   instHMISettings.instAsnBtnPrms.settings.stations.nextGroup.animate := 4;
   instHMISettings.instAsnBtnPrms.settings.stations.prevGroup.animate := 4;
   instHMISettings.instAsnBtnPrms.settings.stations.selectBtns[0].animate := 4;
   instHMISettings.instAsnBtnPrms.settings.stations.selectBtns[0].label := WSTRING#'1BX 3.0 1';
   instHMISettings.instAsnBtnPrms.settings.stations.selectBtns[1].animate := 4;
   instHMISettings.instAsnBtnPrms.settings.stations.selectBtns[1].label := WSTRING#'1BX 3.0 2';
   instHMISettings.instAsnBtnPrms.settings.stations.selectBtns[2].animate := 4;
   instHMISettings.instAsnBtnPrms.settings.stations.selectBtns[2].label := WSTRING#'1BX 3.0 3';
   instHMISettings.instAsnBtnPrms.settings.stations.selectBtns[3].animate := 4;
   instHMISettings.instAsnBtnPrms.settings.stations.selectBtns[3].label := WSTRING#'VOLVO 16 1';
   instHMISettings.instAsnBtnPrms.settings.stations.selectBtns[4].animate := 4;
   instHMISettings.instAsnBtnPrms.settings.stations.selectBtns[4].label := WSTRING#'VOLVO 16 2';
   instHMISettings.instAsnBtnPrms.settings.stations.selectBtns[5].animate := 4;
   instHMISettings.instAsnBtnPrms.settings.stations.selectBtns[5].label := WSTRING#'VOLVO 16 3';
   instHMISettings.instAsnBtnPrms.settings.stations.selectBtns[6].animate := 4;
   instHMISettings.instAsnBtnPrms.settings.stations.selectBtns[6].label := WSTRING#'VOLVO 16 4';
   instHMISettings.instAsnBtnPrms.settings.stations.selectBtns[7].animate := 4;
   instHMISettings.instAsnBtnPrms.settings.stations.selectBtns[7].label := WSTRING#'VOLVO 16 5';
   instHMISettings.instAsnBtnPrms.settings.stations.selectBtns[8].animate := 4;
   instHMISettings.instAsnBtnPrms.settings.stations.selectBtns[8].label := WSTRING#'VOLVO 16 6';
   instHMISettings.instAsnBtnPrms.settings.stations.selectBtns[9].animate := 4;
   instHMISettings.instAsnBtnPrms.settings.stations.selectBtns[9].label := WSTRING#'VOLVO 16 7';
   instHMISettings.instAsnBtnPrms.settings.stations.selectBtns[10].animate := 4;
   instHMISettings.instAsnBtnPrms.settings.stations.selectBtns[10].label := WSTRING#'VOLVO 16 8';
   instHMISettings.instAsnBtnPrms.settings.stations.selectBtns[11].animate := 4;
   instHMISettings.instAsnBtnPrms.settings.stations.selectBtns[11].label := WSTRING#'VOLVO 16 9';
   instHMISettings.instAsnBtnPrms.settings.stations.selCount := 1;
   instHMISettings.instAsnBtnPrms.settings.stations.selNumber := 19;
   instHMISettings.instAsnBtnPrms.settings.partNumber.assign.animate := 254;
   instHMISettings.instAsnBtnPrms.settings.partNumber.assign.label := WSTRING#'';
   instHMISettings.instAsnBtnPrms.settings.partNumber.ioField.animate := 254;
   instHMISettings.instAsnBtnPrms.settings.partNumber.ioField.inputFinished := TRUE;
   instHMISettings.instAsnBtnPrms.settings.partNumber.ioField.value := WSTRING#'';
   instHMISettings.instAsnBtnPrms.settings.viewingStation.btns[0].alloted.animate := 4;
   instHMISettings.instAsnBtnPrms.settings.viewingStation.btns[0].alloted.value := WSTRING#'30:00';
   instHMISettings.instAsnBtnPrms.settings.viewingStation.btns[0].critical.animate := 4;
   instHMISettings.instAsnBtnPrms.settings.viewingStation.btns[0].critical.value := WSTRING#'05:00';
   instHMISettings.instAsnBtnPrms.settings.viewingStation.btns[0].label.animate := 4;
   instHMISettings.instAsnBtnPrms.settings.viewingStation.btns[0].label.value := WSTRING#'1';
   instHMISettings.instAsnBtnPrms.settings.viewingStation.btns[0].partNumber.animate := 4;
   instHMISettings.instAsnBtnPrms.settings.viewingStation.btns[0].partNumber.value := WSTRING#'16.08.211.511.020F';
   instHMISettings.instAsnBtnPrms.settings.viewingStation.btns[1].alloted.animate := 4;
   instHMISettings.instAsnBtnPrms.settings.viewingStation.btns[1].alloted.value := WSTRING#'30:00';
   instHMISettings.instAsnBtnPrms.settings.viewingStation.btns[1].critical.animate := 4;
   instHMISettings.instAsnBtnPrms.settings.viewingStation.btns[1].critical.value := WSTRING#'05:00';
   instHMISettings.instAsnBtnPrms.settings.viewingStation.btns[1].label.animate := 4;
   instHMISettings.instAsnBtnPrms.settings.viewingStation.btns[1].label.value := WSTRING#'2';
   instHMISettings.instAsnBtnPrms.settings.viewingStation.btns[1].partNumber.animate := 4;
   instHMISettings.instAsnBtnPrms.settings.viewingStation.btns[1].partNumber.value := WSTRING#'16.08.208.151.010F';
   instHMISettings.instAsnBtnPrms.settings.viewingStation.btns[2].alloted.animate := 4;
   instHMISettings.instAsnBtnPrms.settings.viewingStation.btns[2].alloted.value := WSTRING#'30:00';
   instHMISettings.instAsnBtnPrms.settings.viewingStation.btns[2].critical.animate := 4;
   instHMISettings.instAsnBtnPrms.settings.viewingStation.btns[2].critical.value := WSTRING#'05:00';
   instHMISettings.instAsnBtnPrms.settings.viewingStation.btns[2].label.animate := 4;
   instHMISettings.instAsnBtnPrms.settings.viewingStation.btns[2].label.value := WSTRING#'3';
   instHMISettings.instAsnBtnPrms.settings.viewingStation.btns[2].partNumber.animate := 4;
   instHMISettings.instAsnBtnPrms.settings.viewingStation.btns[2].partNumber.value := WSTRING#'16.08.216.151.010B';
   instHMISettings.instAsnBtnPrms.settings.viewingStation.btns[3].alloted.animate := 4;
   instHMISettings.instAsnBtnPrms.settings.viewingStation.btns[3].alloted.value := WSTRING#'30:00';
   instHMISettings.instAsnBtnPrms.settings.viewingStation.btns[3].critical.animate := 4;
   instHMISettings.instAsnBtnPrms.settings.viewingStation.btns[3].critical.value := WSTRING#'05:00';
   instHMISettings.instAsnBtnPrms.settings.viewingStation.btns[3].label.animate := 4;
   instHMISettings.instAsnBtnPrms.settings.viewingStation.btns[3].label.value := WSTRING#'4';
   instHMISettings.instAsnBtnPrms.settings.viewingStation.btns[3].partNumber.animate := 4;
   instHMISettings.instAsnBtnPrms.settings.viewingStation.btns[3].partNumber.value := WSTRING#'16.08.216.831.020A';
   instHMISettings.instAsnBtnPrms.settings.viewingStation.btns[4].alloted.animate := 4;
   instHMISettings.instAsnBtnPrms.settings.viewingStation.btns[4].alloted.value := WSTRING#'02:00';
   instHMISettings.instAsnBtnPrms.settings.viewingStation.btns[4].critical.animate := 4;
   instHMISettings.instAsnBtnPrms.settings.viewingStation.btns[4].critical.value := WSTRING#'01:10';
   instHMISettings.instAsnBtnPrms.settings.viewingStation.btns[4].label.animate := 4;
   instHMISettings.instAsnBtnPrms.settings.viewingStation.btns[4].label.value := WSTRING#'5';
   instHMISettings.instAsnBtnPrms.settings.viewingStation.btns[4].partNumber.animate := 4;
   instHMISettings.instAsnBtnPrms.settings.viewingStation.btns[4].partNumber.value := WSTRING#'16.08.217.411.080A';
   instHMISettings.instAsnBtnPrms.settings.viewingStation.btns[5].alloted.animate := 4;
   instHMISettings.instAsnBtnPrms.settings.viewingStation.btns[5].alloted.value := WSTRING#'30:00';
   instHMISettings.instAsnBtnPrms.settings.viewingStation.btns[5].critical.animate := 4;
   instHMISettings.instAsnBtnPrms.settings.viewingStation.btns[5].critical.value := WSTRING#'05:00';
   instHMISettings.instAsnBtnPrms.settings.viewingStation.btns[5].label.animate := 4;
   instHMISettings.instAsnBtnPrms.settings.viewingStation.btns[5].label.value := WSTRING#'6';
   instHMISettings.instAsnBtnPrms.settings.viewingStation.btns[5].partNumber.animate := 4;
   instHMISettings.instAsnBtnPrms.settings.viewingStation.btns[5].partNumber.value := WSTRING#'16.08.216.521.000F';
   instHMISettings.instAsnBtnPrms.settings.viewingStation.btns[6].alloted.animate := 4;
   instHMISettings.instAsnBtnPrms.settings.viewingStation.btns[6].alloted.value := WSTRING#'00:00';
   instHMISettings.instAsnBtnPrms.settings.viewingStation.btns[6].critical.animate := 4;
   instHMISettings.instAsnBtnPrms.settings.viewingStation.btns[6].critical.value := WSTRING#'00:00';
   instHMISettings.instAsnBtnPrms.settings.viewingStation.btns[6].label.animate := 4;
   instHMISettings.instAsnBtnPrms.settings.viewingStation.btns[6].label.value := WSTRING#'7';
   instHMISettings.instAsnBtnPrms.settings.viewingStation.btns[6].partNumber.animate := 4;
   instHMISettings.instAsnBtnPrms.settings.viewingStation.btns[6].partNumber.value := WSTRING#'';
   instHMISettings.instAsnBtnPrms.settings.viewingStation.btns[7].alloted.animate := 4;
   instHMISettings.instAsnBtnPrms.settings.viewingStation.btns[7].alloted.value := WSTRING#'00:00';
   instHMISettings.instAsnBtnPrms.settings.viewingStation.btns[7].critical.animate := 4;
   instHMISettings.instAsnBtnPrms.settings.viewingStation.btns[7].critical.value := WSTRING#'00:00';
   instHMISettings.instAsnBtnPrms.settings.viewingStation.btns[7].label.animate := 4;
   instHMISettings.instAsnBtnPrms.settings.viewingStation.btns[7].label.value := WSTRING#'8';
   instHMISettings.instAsnBtnPrms.settings.viewingStation.btns[7].partNumber.animate := 4;
   instHMISettings.instAsnBtnPrms.settings.viewingStation.btns[7].partNumber.value := WSTRING#'';
   instHMISettings.instAsnBtnPrms.settings.viewingStation.dzData.animate.bg := 4;
   instHMISettings.instAsnBtnPrms.settings.viewingStation.dzData.animate.ioField := 1;
   instHMISettings.instAsnBtnPrms.settings.viewingStation.dzData.value := WSTRING#'1';
   instHMISettings.instAsnBtnPrms.settings.viewingStation.lineData.animate.bg := 4;
   instHMISettings.instAsnBtnPrms.settings.viewingStation.lineData.animate.ioField := 1;
   instHMISettings.instAsnBtnPrms.settings.viewingStation.lineData.value := WSTRING#'BFL';
   instHMISettings.instAsnBtnPrms.settings.viewingStation.next.animate := 4;
   instHMISettings.instAsnBtnPrms.settings.viewingStation.previous.animate := 4;
   instHMISettings.instAsnBtnPrms.settings.viewingStation."name" := WSTRING#'BFL 1';
   instHMISettings.instAniPNTmr.stations.me[0].dropZone := 1;
   instHMISettings.instAniPNTmr.stations.me[0].kp8Config.activate[3] := TRUE;
   instHMISettings.instAniPNTmr.stations.me[0].kp8Config.activate[7] := TRUE;
   instHMISettings.instAniPNTmr.stations.me[0].kp8Config.colorOn1[0] := 'off';
   instHMISettings.instAniPNTmr.stations.me[0].kp8Config.colorOn1[1] := 'off';
   instHMISettings.instAniPNTmr.stations.me[0].kp8Config.colorOn1[2] := 'off';
   instHMISettings.instAniPNTmr.stations.me[0].kp8Config.colorOn1[3] := 'yellow';
   instHMISettings.instAniPNTmr.stations.me[0].kp8Config.colorOn1[4] := 'off';
   instHMISettings.instAniPNTmr.stations.me[0].kp8Config.colorOn1[5] := 'off';
   instHMISettings.instAniPNTmr.stations.me[0].kp8Config.colorOn1[6] := 'off';
   instHMISettings.instAniPNTmr.stations.me[0].kp8Config.colorOn1[7] := 'yellow';
   instHMISettings.instAniPNTmr.stations.me[0].kp8Config.colorOn2[0] := 'off';
   instHMISettings.instAniPNTmr.stations.me[0].kp8Config.colorOn2[1] := 'off';
   instHMISettings.instAniPNTmr.stations.me[0].kp8Config.colorOn2[2] := 'off';
   instHMISettings.instAniPNTmr.stations.me[0].kp8Config.colorOn2[4] := 'off';
   instHMISettings.instAniPNTmr.stations.me[0].kp8Config.colorOn2[5] := 'off';
   instHMISettings.instAniPNTmr.stations.me[0].kp8Config.colorOn2[6] := 'off';
   instHMISettings.instAniPNTmr.stations.me[0].kp8Config.colorOff[0] := 'off';
   instHMISettings.instAniPNTmr.stations.me[0].kp8Config.colorOff[1] := 'off';
   instHMISettings.instAniPNTmr.stations.me[0].kp8Config.colorOff[2] := 'off';
   instHMISettings.instAniPNTmr.stations.me[0].kp8Config.colorOff[3] := 'green';
   instHMISettings.instAniPNTmr.stations.me[0].kp8Config.colorOff[4] := 'off';
   instHMISettings.instAniPNTmr.stations.me[0].kp8Config.colorOff[5] := 'off';
   instHMISettings.instAniPNTmr.stations.me[0].kp8Config.colorOff[6] := 'off';
   instHMISettings.instAniPNTmr.stations.me[0].kp8Config.colorOff[7] := 'green';
   instHMISettings.instAniPNTmr.stations.me[0].kp8Config.mode[3] := TRUE;
   instHMISettings.instAniPNTmr.stations.me[0].kp8Config.mode[7] := TRUE;
   instHMISettings.instAniPNTmr.stations.me[0].kp8Out := 16#0088_0000;
   instHMISettings.instAniPNTmr.stations.me[0].line := WSTRING#'VOLVO 16';
   instHMISettings.instAniPNTmr.stations.me[0].partNumbers[0] := WSTRING#'';
   instHMISettings.instAniPNTmr.stations.me[0].partNumbers[1] := WSTRING#'';
   instHMISettings.instAniPNTmr.stations.me[0].partNumbers[2] := WSTRING#'';
   instHMISettings.instAniPNTmr.stations.me[0].partNumbers[3] := WSTRING#'16.32.112.500.220A';
   instHMISettings.instAniPNTmr.stations.me[0].partNumbers[4] := WSTRING#'';
   instHMISettings.instAniPNTmr.stations.me[0].partNumbers[5] := WSTRING#'';
   instHMISettings.instAniPNTmr.stations.me[0].partNumbers[6] := WSTRING#'';
   instHMISettings.instAniPNTmr.stations.me[0].partNumbers[7] := WSTRING#'16.32.112.500.100A';
   instHMISettings.instAniPNTmr.stations.me[0].presetTime.allotted[3] := 1800.0;
   instHMISettings.instAniPNTmr.stations.me[0].presetTime.allotted[7] := 1800.0;
   instHMISettings.instAniPNTmr.stations.me[0].presetTime.critical[3] := 300.0;
   instHMISettings.instAniPNTmr.stations.me[0].presetTime.critical[7] := 300.0;
   instHMISettings.instAniPNTmr.stations.me[0].stackLightOut := 16#2400_0000;
   instHMISettings.instAniPNTmr.stations.me[1].dropZone := 2;
   instHMISettings.instAniPNTmr.stations.me[1].kp8Config.activate[2] := TRUE;
   instHMISettings.instAniPNTmr.stations.me[1].kp8Config.activate[3] := TRUE;
   instHMISettings.instAniPNTmr.stations.me[1].kp8Config.activate[6] := TRUE;
   instHMISettings.instAniPNTmr.stations.me[1].kp8Config.activate[7] := TRUE;
   instHMISettings.instAniPNTmr.stations.me[1].kp8Config.colorOn1[0] := 'off';
   instHMISettings.instAniPNTmr.stations.me[1].kp8Config.colorOn1[1] := 'off';
   instHMISettings.instAniPNTmr.stations.me[1].kp8Config.colorOn1[2] := 'yellow';
   instHMISettings.instAniPNTmr.stations.me[1].kp8Config.colorOn1[3] := 'yellow';
   instHMISettings.instAniPNTmr.stations.me[1].kp8Config.colorOn1[4] := 'off';
   instHMISettings.instAniPNTmr.stations.me[1].kp8Config.colorOn1[5] := 'off';
   instHMISettings.instAniPNTmr.stations.me[1].kp8Config.colorOn1[6] := 'yellow';
   instHMISettings.instAniPNTmr.stations.me[1].kp8Config.colorOn1[7] := 'yellow';
   instHMISettings.instAniPNTmr.stations.me[1].kp8Config.colorOn2[0] := 'off';
   instHMISettings.instAniPNTmr.stations.me[1].kp8Config.colorOn2[1] := 'off';
   instHMISettings.instAniPNTmr.stations.me[1].kp8Config.colorOn2[4] := 'off';
   instHMISettings.instAniPNTmr.stations.me[1].kp8Config.colorOn2[5] := 'off';
   instHMISettings.instAniPNTmr.stations.me[1].kp8Config.colorOff[0] := 'off';
   instHMISettings.instAniPNTmr.stations.me[1].kp8Config.colorOff[1] := 'off';
   instHMISettings.instAniPNTmr.stations.me[1].kp8Config.colorOff[2] := 'green';
   instHMISettings.instAniPNTmr.stations.me[1].kp8Config.colorOff[3] := 'green';
   instHMISettings.instAniPNTmr.stations.me[1].kp8Config.colorOff[4] := 'off';
   instHMISettings.instAniPNTmr.stations.me[1].kp8Config.colorOff[5] := 'off';
   instHMISettings.instAniPNTmr.stations.me[1].kp8Config.colorOff[6] := 'green';
   instHMISettings.instAniPNTmr.stations.me[1].kp8Config.colorOff[7] := 'green';
   instHMISettings.instAniPNTmr.stations.me[1].kp8Config.mode[2] := TRUE;
   instHMISettings.instAniPNTmr.stations.me[1].kp8Config.mode[3] := TRUE;
   instHMISettings.instAniPNTmr.stations.me[1].kp8Config.mode[6] := TRUE;
   instHMISettings.instAniPNTmr.stations.me[1].kp8Config.mode[7] := TRUE;
   instHMISettings.instAniPNTmr.stations.me[1].kp8Out := 16#00CC_0000;
   instHMISettings.instAniPNTmr.stations.me[1].line := WSTRING#'VOLVO 16';
   instHMISettings.instAniPNTmr.stations.me[1].partNumbers[0] := WSTRING#'';
   instHMISettings.instAniPNTmr.stations.me[1].partNumbers[1] := WSTRING#'';
   instHMISettings.instAniPNTmr.stations.me[1].partNumbers[2] := WSTRING#'16.32.112.509.070A';
   instHMISettings.instAniPNTmr.stations.me[1].partNumbers[3] := WSTRING#'16.32.112.704.000C';
   instHMISettings.instAniPNTmr.stations.me[1].partNumbers[4] := WSTRING#'';
   instHMISettings.instAniPNTmr.stations.me[1].partNumbers[5] := WSTRING#'';
   instHMISettings.instAniPNTmr.stations.me[1].partNumbers[6] := WSTRING#'16.32.112.504.060A';
   instHMISettings.instAniPNTmr.stations.me[1].partNumbers[7] := WSTRING#'16.32.112.500.060D';
   instHMISettings.instAniPNTmr.stations.me[1].presetTime.allotted[2] := 1800.0;
   instHMISettings.instAniPNTmr.stations.me[1].presetTime.allotted[3] := 1800.0;
   instHMISettings.instAniPNTmr.stations.me[1].presetTime.allotted[6] := 1800.0;
   instHMISettings.instAniPNTmr.stations.me[1].presetTime.allotted[7] := 1800.0;
   instHMISettings.instAniPNTmr.stations.me[1].presetTime.critical[2] := 300.0;
   instHMISettings.instAniPNTmr.stations.me[1].presetTime.critical[3] := 300.0;
   instHMISettings.instAniPNTmr.stations.me[1].presetTime.critical[6] := 300.0;
   instHMISettings.instAniPNTmr.stations.me[1].presetTime.critical[7] := 300.0;
   instHMISettings.instAniPNTmr.stations.me[1].stackLightOut := 16#2409_0000;
   instHMISettings.instAniPNTmr.stations.me[2].dropZone := 3;
   instHMISettings.instAniPNTmr.stations.me[2].kp8Config.activate[1] := TRUE;
   instHMISettings.instAniPNTmr.stations.me[2].kp8Config.activate[2] := TRUE;
   instHMISettings.instAniPNTmr.stations.me[2].kp8Config.activate[3] := TRUE;
   instHMISettings.instAniPNTmr.stations.me[2].kp8Config.activate[5] := TRUE;
   instHMISettings.instAniPNTmr.stations.me[2].kp8Config.activate[6] := TRUE;
   instHMISettings.instAniPNTmr.stations.me[2].kp8Config.activate[7] := TRUE;
   instHMISettings.instAniPNTmr.stations.me[2].kp8Config.colorOn1[0] := 'off';
   instHMISettings.instAniPNTmr.stations.me[2].kp8Config.colorOn1[1] := 'yellow';
   instHMISettings.instAniPNTmr.stations.me[2].kp8Config.colorOn1[2] := 'yellow';
   instHMISettings.instAniPNTmr.stations.me[2].kp8Config.colorOn1[3] := 'yellow';
   instHMISettings.instAniPNTmr.stations.me[2].kp8Config.colorOn1[4] := 'off';
   instHMISettings.instAniPNTmr.stations.me[2].kp8Config.colorOn1[5] := 'yellow';
   instHMISettings.instAniPNTmr.stations.me[2].kp8Config.colorOn1[6] := 'yellow';
   instHMISettings.instAniPNTmr.stations.me[2].kp8Config.colorOn1[7] := 'yellow';
   instHMISettings.instAniPNTmr.stations.me[2].kp8Config.colorOn2[0] := 'off';
   instHMISettings.instAniPNTmr.stations.me[2].kp8Config.colorOn2[4] := 'off';
   instHMISettings.instAniPNTmr.stations.me[2].kp8Config.colorOff[0] := 'off';
   instHMISettings.instAniPNTmr.stations.me[2].kp8Config.colorOff[1] := 'green';
   instHMISettings.instAniPNTmr.stations.me[2].kp8Config.colorOff[2] := 'green';
   instHMISettings.instAniPNTmr.stations.me[2].kp8Config.colorOff[3] := 'green';
   instHMISettings.instAniPNTmr.stations.me[2].kp8Config.colorOff[4] := 'off';
   instHMISettings.instAniPNTmr.stations.me[2].kp8Config.colorOff[5] := 'green';
   instHMISettings.instAniPNTmr.stations.me[2].kp8Config.colorOff[6] := 'green';
   instHMISettings.instAniPNTmr.stations.me[2].kp8Config.colorOff[7] := 'green';
   instHMISettings.instAniPNTmr.stations.me[2].kp8Config.mode[1] := TRUE;
   instHMISettings.instAniPNTmr.stations.me[2].kp8Config.mode[2] := TRUE;
   instHMISettings.instAniPNTmr.stations.me[2].kp8Config.mode[3] := TRUE;
   instHMISettings.instAniPNTmr.stations.me[2].kp8Config.mode[5] := TRUE;
   instHMISettings.instAniPNTmr.stations.me[2].kp8Config.mode[6] := TRUE;
   instHMISettings.instAniPNTmr.stations.me[2].kp8Config.mode[7] := TRUE;
   instHMISettings.instAniPNTmr.stations.me[2].kp8Out := 16#00EE_0000;
   instHMISettings.instAniPNTmr.stations.me[2].line := WSTRING#'VOLVO 16';
   instHMISettings.instAniPNTmr.stations.me[2].partNumbers[0] := WSTRING#'';
   instHMISettings.instAniPNTmr.stations.me[2].partNumbers[1] := WSTRING#'16.32.112.509.050E';
   instHMISettings.instAniPNTmr.stations.me[2].partNumbers[2] := WSTRING#'16.32.112.504.070G';
   instHMISettings.instAniPNTmr.stations.me[2].partNumbers[3] := WSTRING#'16.32.112.851.001A';
   instHMISettings.instAniPNTmr.stations.me[2].partNumbers[4] := WSTRING#'';
   instHMISettings.instAniPNTmr.stations.me[2].partNumbers[5] := WSTRING#'16.32.112.509.080F';
   instHMISettings.instAniPNTmr.stations.me[2].partNumbers[6] := WSTRING#'16.32.112.870.000C';
   instHMISettings.instAniPNTmr.stations.me[2].partNumbers[7] := WSTRING#'16.32.112.851.000B';
   instHMISettings.instAniPNTmr.stations.me[2].presetTime.allotted[1] := 1800.0;
   instHMISettings.instAniPNTmr.stations.me[2].presetTime.allotted[2] := 1800.0;
   instHMISettings.instAniPNTmr.stations.me[2].presetTime.allotted[3] := 1800.0;
   instHMISettings.instAniPNTmr.stations.me[2].presetTime.allotted[5] := 1800.0;
   instHMISettings.instAniPNTmr.stations.me[2].presetTime.allotted[6] := 1800.0;
   instHMISettings.instAniPNTmr.stations.me[2].presetTime.allotted[7] := 1800.0;
   instHMISettings.instAniPNTmr.stations.me[2].presetTime.critical[1] := 300.0;
   instHMISettings.instAniPNTmr.stations.me[2].presetTime.critical[2] := 300.0;
   instHMISettings.instAniPNTmr.stations.me[2].presetTime.critical[3] := 300.0;
   instHMISettings.instAniPNTmr.stations.me[2].presetTime.critical[5] := 300.0;
   instHMISettings.instAniPNTmr.stations.me[2].presetTime.critical[6] := 300.0;
   instHMISettings.instAniPNTmr.stations.me[2].presetTime.critical[7] := 300.0;
   instHMISettings.instAniPNTmr.stations.me[2].stackLightOut := 16#2449_0200;
   instHMISettings.instAniPNTmr.stations.me[3].dropZone := 4;
   instHMISettings.instAniPNTmr.stations.me[3].kp8Config.activate[1] := TRUE;
   instHMISettings.instAniPNTmr.stations.me[3].kp8Config.activate[2] := TRUE;
   instHMISettings.instAniPNTmr.stations.me[3].kp8Config.activate[3] := TRUE;
   instHMISettings.instAniPNTmr.stations.me[3].kp8Config.activate[5] := TRUE;
   instHMISettings.instAniPNTmr.stations.me[3].kp8Config.activate[6] := TRUE;
   instHMISettings.instAniPNTmr.stations.me[3].kp8Config.activate[7] := TRUE;
   instHMISettings.instAniPNTmr.stations.me[3].kp8Config.colorOn1[0] := 'off';
   instHMISettings.instAniPNTmr.stations.me[3].kp8Config.colorOn1[1] := 'yellow';
   instHMISettings.instAniPNTmr.stations.me[3].kp8Config.colorOn1[2] := 'yellow';
   instHMISettings.instAniPNTmr.stations.me[3].kp8Config.colorOn1[3] := 'yellow';
   instHMISettings.instAniPNTmr.stations.me[3].kp8Config.colorOn1[4] := 'off';
   instHMISettings.instAniPNTmr.stations.me[3].kp8Config.colorOn1[5] := 'yellow';
   instHMISettings.instAniPNTmr.stations.me[3].kp8Config.colorOn1[6] := 'yellow';
   instHMISettings.instAniPNTmr.stations.me[3].kp8Config.colorOn1[7] := 'yellow';
   instHMISettings.instAniPNTmr.stations.me[3].kp8Config.colorOn2[0] := 'off';
   instHMISettings.instAniPNTmr.stations.me[3].kp8Config.colorOn2[4] := 'off';
   instHMISettings.instAniPNTmr.stations.me[3].kp8Config.colorOff[0] := 'off';
   instHMISettings.instAniPNTmr.stations.me[3].kp8Config.colorOff[1] := 'green';
   instHMISettings.instAniPNTmr.stations.me[3].kp8Config.colorOff[2] := 'green';
   instHMISettings.instAniPNTmr.stations.me[3].kp8Config.colorOff[3] := 'green';
   instHMISettings.instAniPNTmr.stations.me[3].kp8Config.colorOff[4] := 'off';
   instHMISettings.instAniPNTmr.stations.me[3].kp8Config.colorOff[5] := 'green';
   instHMISettings.instAniPNTmr.stations.me[3].kp8Config.colorOff[6] := 'green';
   instHMISettings.instAniPNTmr.stations.me[3].kp8Config.colorOff[7] := 'green';
   instHMISettings.instAniPNTmr.stations.me[3].kp8Config.mode[1] := TRUE;
   instHMISettings.instAniPNTmr.stations.me[3].kp8Config.mode[2] := TRUE;
   instHMISettings.instAniPNTmr.stations.me[3].kp8Config.mode[3] := TRUE;
   instHMISettings.instAniPNTmr.stations.me[3].kp8Config.mode[5] := TRUE;
   instHMISettings.instAniPNTmr.stations.me[3].kp8Config.mode[6] := TRUE;
   instHMISettings.instAniPNTmr.stations.me[3].kp8Config.mode[7] := TRUE;
   instHMISettings.instAniPNTmr.stations.me[3].kp8Out := 16#00EE_0000;
   instHMISettings.instAniPNTmr.stations.me[3].line := WSTRING#'VOLVO 16';
   instHMISettings.instAniPNTmr.stations.me[3].partNumbers[0] := WSTRING#'';
   instHMISettings.instAniPNTmr.stations.me[3].partNumbers[1] := WSTRING#'16.32.112.522.130A';
   instHMISettings.instAniPNTmr.stations.me[3].partNumbers[2] := WSTRING#'16.32.112.522.050A';
   instHMISettings.instAniPNTmr.stations.me[3].partNumbers[3] := WSTRING#'16.32.112.521.020B';
   instHMISettings.instAniPNTmr.stations.me[3].partNumbers[4] := WSTRING#'';
   instHMISettings.instAniPNTmr.stations.me[3].partNumbers[5] := WSTRING#'16.32.112.522.040D';
   instHMISettings.instAniPNTmr.stations.me[3].partNumbers[6] := WSTRING#'16.32.112.521.010B';
   instHMISettings.instAniPNTmr.stations.me[3].partNumbers[7] := WSTRING#'16.32.112.521.030A';
   instHMISettings.instAniPNTmr.stations.me[3].presetTime.allotted[1] := 1800.0;
   instHMISettings.instAniPNTmr.stations.me[3].presetTime.allotted[2] := 1800.0;
   instHMISettings.instAniPNTmr.stations.me[3].presetTime.allotted[3] := 1800.0;
   instHMISettings.instAniPNTmr.stations.me[3].presetTime.allotted[5] := 1800.0;
   instHMISettings.instAniPNTmr.stations.me[3].presetTime.allotted[6] := 1800.0;
   instHMISettings.instAniPNTmr.stations.me[3].presetTime.allotted[7] := 1800.0;
   instHMISettings.instAniPNTmr.stations.me[3].presetTime.critical[1] := 300.0;
   instHMISettings.instAniPNTmr.stations.me[3].presetTime.critical[2] := 300.0;
   instHMISettings.instAniPNTmr.stations.me[3].presetTime.critical[3] := 300.0;
   instHMISettings.instAniPNTmr.stations.me[3].presetTime.critical[5] := 300.0;
   instHMISettings.instAniPNTmr.stations.me[3].presetTime.critical[6] := 300.0;
   instHMISettings.instAniPNTmr.stations.me[3].presetTime.critical[7] := 300.0;
   instHMISettings.instAniPNTmr.stations.me[3].stackLightOut := 16#2449_0200;
   instHMISettings.instAniPNTmr.stations.me[4].dropZone := 5;
   instHMISettings.instAniPNTmr.stations.me[4].kp8Config.activate[7] := TRUE;
   instHMISettings.instAniPNTmr.stations.me[4].kp8Config.colorOn1[0] := 'off';
   instHMISettings.instAniPNTmr.stations.me[4].kp8Config.colorOn1[1] := 'off';
   instHMISettings.instAniPNTmr.stations.me[4].kp8Config.colorOn1[2] := 'off';
   instHMISettings.instAniPNTmr.stations.me[4].kp8Config.colorOn1[3] := 'off';
   instHMISettings.instAniPNTmr.stations.me[4].kp8Config.colorOn1[4] := 'off';
   instHMISettings.instAniPNTmr.stations.me[4].kp8Config.colorOn1[5] := 'off';
   instHMISettings.instAniPNTmr.stations.me[4].kp8Config.colorOn1[6] := 'off';
   instHMISettings.instAniPNTmr.stations.me[4].kp8Config.colorOn1[7] := 'yellow';
   instHMISettings.instAniPNTmr.stations.me[4].kp8Config.colorOn2[0] := 'off';
   instHMISettings.instAniPNTmr.stations.me[4].kp8Config.colorOn2[1] := 'off';
   instHMISettings.instAniPNTmr.stations.me[4].kp8Config.colorOn2[2] := 'off';
   instHMISettings.instAniPNTmr.stations.me[4].kp8Config.colorOn2[3] := 'off';
   instHMISettings.instAniPNTmr.stations.me[4].kp8Config.colorOn2[4] := 'off';
   instHMISettings.instAniPNTmr.stations.me[4].kp8Config.colorOn2[5] := 'off';
   instHMISettings.instAniPNTmr.stations.me[4].kp8Config.colorOn2[6] := 'off';
   instHMISettings.instAniPNTmr.stations.me[4].kp8Config.colorOff[0] := 'off';
   instHMISettings.instAniPNTmr.stations.me[4].kp8Config.colorOff[1] := 'off';
   instHMISettings.instAniPNTmr.stations.me[4].kp8Config.colorOff[2] := 'off';
   instHMISettings.instAniPNTmr.stations.me[4].kp8Config.colorOff[3] := 'off';
   instHMISettings.instAniPNTmr.stations.me[4].kp8Config.colorOff[4] := 'off';
   instHMISettings.instAniPNTmr.stations.me[4].kp8Config.colorOff[5] := 'off';
   instHMISettings.instAniPNTmr.stations.me[4].kp8Config.colorOff[6] := 'off';
   instHMISettings.instAniPNTmr.stations.me[4].kp8Config.colorOff[7] := 'green';
   instHMISettings.instAniPNTmr.stations.me[4].kp8Config.mode[7] := TRUE;
   instHMISettings.instAniPNTmr.stations.me[4].kp8Out := 16#0080_0000;
   instHMISettings.instAniPNTmr.stations.me[4].line := WSTRING#'VOLVO 16';
   instHMISettings.instAniPNTmr.stations.me[4].partNumbers[0] := WSTRING#'';
   instHMISettings.instAniPNTmr.stations.me[4].partNumbers[1] := WSTRING#'';
   instHMISettings.instAniPNTmr.stations.me[4].partNumbers[2] := WSTRING#'';
   instHMISettings.instAniPNTmr.stations.me[4].partNumbers[3] := WSTRING#'';
   instHMISettings.instAniPNTmr.stations.me[4].partNumbers[4] := WSTRING#'';
   instHMISettings.instAniPNTmr.stations.me[4].partNumbers[5] := WSTRING#'';
   instHMISettings.instAniPNTmr.stations.me[4].partNumbers[6] := WSTRING#'';
   instHMISettings.instAniPNTmr.stations.me[4].partNumbers[7] := WSTRING#'16.32.112.529.020B';
   instHMISettings.instAniPNTmr.stations.me[4].presetTime.allotted[7] := 1800.0;
   instHMISettings.instAniPNTmr.stations.me[4].presetTime.critical[7] := 300.0;
   instHMISettings.instAniPNTmr.stations.me[4].stackLightOut := 16#0400_0000;
   instHMISettings.instAniPNTmr.stations.me[5].dropZone := 6;
   instHMISettings.instAniPNTmr.stations.me[5].kp8Config.activate[1] := TRUE;
   instHMISettings.instAniPNTmr.stations.me[5].kp8Config.activate[2] := TRUE;
   instHMISettings.instAniPNTmr.stations.me[5].kp8Config.activate[3] := TRUE;
   instHMISettings.instAniPNTmr.stations.me[5].kp8Config.activate[5] := TRUE;
   instHMISettings.instAniPNTmr.stations.me[5].kp8Config.activate[6] := TRUE;
   instHMISettings.instAniPNTmr.stations.me[5].kp8Config.activate[7] := TRUE;
   instHMISettings.instAniPNTmr.stations.me[5].kp8Config.colorOn1[0] := 'off';
   instHMISettings.instAniPNTmr.stations.me[5].kp8Config.colorOn1[1] := 'yellow';
   instHMISettings.instAniPNTmr.stations.me[5].kp8Config.colorOn1[2] := 'yellow';
   instHMISettings.instAniPNTmr.stations.me[5].kp8Config.colorOn1[3] := 'yellow';
   instHMISettings.instAniPNTmr.stations.me[5].kp8Config.colorOn1[4] := 'off';
   instHMISettings.instAniPNTmr.stations.me[5].kp8Config.colorOn1[5] := 'yellow';
   instHMISettings.instAniPNTmr.stations.me[5].kp8Config.colorOn1[6] := 'yellow';
   instHMISettings.instAniPNTmr.stations.me[5].kp8Config.colorOn1[7] := 'yellow';
   instHMISettings.instAniPNTmr.stations.me[5].kp8Config.colorOn2[0] := 'off';
   instHMISettings.instAniPNTmr.stations.me[5].kp8Config.colorOn2[4] := 'off';
   instHMISettings.instAniPNTmr.stations.me[5].kp8Config.colorOff[0] := 'off';
   instHMISettings.instAniPNTmr.stations.me[5].kp8Config.colorOff[1] := 'green';
   instHMISettings.instAniPNTmr.stations.me[5].kp8Config.colorOff[2] := 'green';
   instHMISettings.instAniPNTmr.stations.me[5].kp8Config.colorOff[3] := 'green';
   instHMISettings.instAniPNTmr.stations.me[5].kp8Config.colorOff[4] := 'off';
   instHMISettings.instAniPNTmr.stations.me[5].kp8Config.colorOff[5] := 'green';
   instHMISettings.instAniPNTmr.stations.me[5].kp8Config.colorOff[6] := 'green';
   instHMISettings.instAniPNTmr.stations.me[5].kp8Config.colorOff[7] := 'green';
   instHMISettings.instAniPNTmr.stations.me[5].kp8Config.mode[1] := TRUE;
   instHMISettings.instAniPNTmr.stations.me[5].kp8Config.mode[2] := TRUE;
   instHMISettings.instAniPNTmr.stations.me[5].kp8Config.mode[3] := TRUE;
   instHMISettings.instAniPNTmr.stations.me[5].kp8Config.mode[5] := TRUE;
   instHMISettings.instAniPNTmr.stations.me[5].kp8Config.mode[6] := TRUE;
   instHMISettings.instAniPNTmr.stations.me[5].kp8Config.mode[7] := TRUE;
   instHMISettings.instAniPNTmr.stations.me[5].kp8Out := 16#00EE_0000;
   instHMISettings.instAniPNTmr.stations.me[5].line := WSTRING#'VOLVO 16';
   instHMISettings.instAniPNTmr.stations.me[5].partNumbers[0] := WSTRING#'';
   instHMISettings.instAniPNTmr.stations.me[5].partNumbers[1] := WSTRING#'16.32.112.529.010A';
   instHMISettings.instAniPNTmr.stations.me[5].partNumbers[2] := WSTRING#'16.32.112.529.030A';
   instHMISettings.instAniPNTmr.stations.me[5].partNumbers[3] := WSTRING#'16.32.112.502.060B';
   instHMISettings.instAniPNTmr.stations.me[5].partNumbers[4] := WSTRING#'';
   instHMISettings.instAniPNTmr.stations.me[5].partNumbers[5] := WSTRING#'16.32.112.529.050D';
   instHMISettings.instAniPNTmr.stations.me[5].partNumbers[6] := WSTRING#'16.32.112.502.070E';
   instHMISettings.instAniPNTmr.stations.me[5].partNumbers[7] := WSTRING#'16.32.112.502.050B';
   instHMISettings.instAniPNTmr.stations.me[5].presetTime.allotted[1] := 1800.0;
   instHMISettings.instAniPNTmr.stations.me[5].presetTime.allotted[2] := 1800.0;
   instHMISettings.instAniPNTmr.stations.me[5].presetTime.allotted[3] := 1800.0;
   instHMISettings.instAniPNTmr.stations.me[5].presetTime.allotted[5] := 1800.0;
   instHMISettings.instAniPNTmr.stations.me[5].presetTime.allotted[6] := 1800.0;
   instHMISettings.instAniPNTmr.stations.me[5].presetTime.allotted[7] := 1800.0;
   instHMISettings.instAniPNTmr.stations.me[5].presetTime.critical[1] := 300.0;
   instHMISettings.instAniPNTmr.stations.me[5].presetTime.critical[2] := 300.0;
   instHMISettings.instAniPNTmr.stations.me[5].presetTime.critical[3] := 300.0;
   instHMISettings.instAniPNTmr.stations.me[5].presetTime.critical[5] := 300.0;
   instHMISettings.instAniPNTmr.stations.me[5].presetTime.critical[6] := 300.0;
   instHMISettings.instAniPNTmr.stations.me[5].presetTime.critical[7] := 300.0;
   instHMISettings.instAniPNTmr.stations.me[5].stackLightOut := 16#2449_0200;
   instHMISettings.instAniPNTmr.stations.me[6].dropZone := 7;
   instHMISettings.instAniPNTmr.stations.me[6].kp8Config.activate[1] := TRUE;
   instHMISettings.instAniPNTmr.stations.me[6].kp8Config.activate[2] := TRUE;
   instHMISettings.instAniPNTmr.stations.me[6].kp8Config.activate[3] := TRUE;
   instHMISettings.instAniPNTmr.stations.me[6].kp8Config.activate[5] := TRUE;
   instHMISettings.instAniPNTmr.stations.me[6].kp8Config.activate[6] := TRUE;
   instHMISettings.instAniPNTmr.stations.me[6].kp8Config.activate[7] := TRUE;
   instHMISettings.instAniPNTmr.stations.me[6].kp8Config.colorOn1[0] := 'off';
   instHMISettings.instAniPNTmr.stations.me[6].kp8Config.colorOn1[1] := 'yellow';
   instHMISettings.instAniPNTmr.stations.me[6].kp8Config.colorOn1[2] := 'yellow';
   instHMISettings.instAniPNTmr.stations.me[6].kp8Config.colorOn1[3] := 'yellow';
   instHMISettings.instAniPNTmr.stations.me[6].kp8Config.colorOn1[4] := 'off';
   instHMISettings.instAniPNTmr.stations.me[6].kp8Config.colorOn1[5] := 'yellow';
   instHMISettings.instAniPNTmr.stations.me[6].kp8Config.colorOn1[6] := 'yellow';
   instHMISettings.instAniPNTmr.stations.me[6].kp8Config.colorOn1[7] := 'yellow';
   instHMISettings.instAniPNTmr.stations.me[6].kp8Config.colorOn2[0] := 'off';
   instHMISettings.instAniPNTmr.stations.me[6].kp8Config.colorOn2[4] := 'off';
   instHMISettings.instAniPNTmr.stations.me[6].kp8Config.colorOff[0] := 'off';
   instHMISettings.instAniPNTmr.stations.me[6].kp8Config.colorOff[1] := 'green';
   instHMISettings.instAniPNTmr.stations.me[6].kp8Config.colorOff[2] := 'green';
   instHMISettings.instAniPNTmr.stations.me[6].kp8Config.colorOff[3] := 'green';
   instHMISettings.instAniPNTmr.stations.me[6].kp8Config.colorOff[4] := 'off';
   instHMISettings.instAniPNTmr.stations.me[6].kp8Config.colorOff[5] := 'green';
   instHMISettings.instAniPNTmr.stations.me[6].kp8Config.colorOff[6] := 'green';
   instHMISettings.instAniPNTmr.stations.me[6].kp8Config.colorOff[7] := 'green';
   instHMISettings.instAniPNTmr.stations.me[6].kp8Config.mode[1] := TRUE;
   instHMISettings.instAniPNTmr.stations.me[6].kp8Config.mode[2] := TRUE;
   instHMISettings.instAniPNTmr.stations.me[6].kp8Config.mode[3] := TRUE;
   instHMISettings.instAniPNTmr.stations.me[6].kp8Config.mode[5] := TRUE;
   instHMISettings.instAniPNTmr.stations.me[6].kp8Config.mode[6] := TRUE;
   instHMISettings.instAniPNTmr.stations.me[6].kp8Config.mode[7] := TRUE;
   instHMISettings.instAniPNTmr.stations.me[6].kp8Out := 16#00EE_0000;
   instHMISettings.instAniPNTmr.stations.me[6].line := WSTRING#'VOLVO 16';
   instHMISettings.instAniPNTmr.stations.me[6].partNumbers[0] := WSTRING#'';
   instHMISettings.instAniPNTmr.stations.me[6].partNumbers[1] := WSTRING#'16.32.112.621.020A';
   instHMISettings.instAniPNTmr.stations.me[6].partNumbers[2] := WSTRING#'16.32.112.621.010A';
   instHMISettings.instAniPNTmr.stations.me[6].partNumbers[3] := WSTRING#'16.32.112.751.000D';
   instHMISettings.instAniPNTmr.stations.me[6].partNumbers[4] := WSTRING#'';
   instHMISettings.instAniPNTmr.stations.me[6].partNumbers[5] := WSTRING#'16.32.112.751.001C';
   instHMISettings.instAniPNTmr.stations.me[6].partNumbers[6] := WSTRING#'16.32.112.601.040A';
   instHMISettings.instAniPNTmr.stations.me[6].partNumbers[7] := WSTRING#'16.32.112.601.030A';
   instHMISettings.instAniPNTmr.stations.me[6].presetTime.allotted[1] := 1800.0;
   instHMISettings.instAniPNTmr.stations.me[6].presetTime.allotted[2] := 1800.0;
   instHMISettings.instAniPNTmr.stations.me[6].presetTime.allotted[3] := 1800.0;
   instHMISettings.instAniPNTmr.stations.me[6].presetTime.allotted[5] := 1800.0;
   instHMISettings.instAniPNTmr.stations.me[6].presetTime.allotted[6] := 1800.0;
   instHMISettings.instAniPNTmr.stations.me[6].presetTime.allotted[7] := 1800.0;
   instHMISettings.instAniPNTmr.stations.me[6].presetTime.critical[1] := 300.0;
   instHMISettings.instAniPNTmr.stations.me[6].presetTime.critical[2] := 300.0;
   instHMISettings.instAniPNTmr.stations.me[6].presetTime.critical[3] := 300.0;
   instHMISettings.instAniPNTmr.stations.me[6].presetTime.critical[5] := 300.0;
   instHMISettings.instAniPNTmr.stations.me[6].presetTime.critical[6] := 300.0;
   instHMISettings.instAniPNTmr.stations.me[6].presetTime.critical[7] := 300.0;
   instHMISettings.instAniPNTmr.stations.me[6].stackLightOut := 16#2449_0200;
   instHMISettings.instAniPNTmr.stations.me[7].dropZone := 8;
   instHMISettings.instAniPNTmr.stations.me[7].kp8Config.activate[3] := TRUE;
   instHMISettings.instAniPNTmr.stations.me[7].kp8Config.activate[6] := TRUE;
   instHMISettings.instAniPNTmr.stations.me[7].kp8Config.activate[7] := TRUE;
   instHMISettings.instAniPNTmr.stations.me[7].kp8Config.colorOn1[0] := 'off';
   instHMISettings.instAniPNTmr.stations.me[7].kp8Config.colorOn1[1] := 'off';
   instHMISettings.instAniPNTmr.stations.me[7].kp8Config.colorOn1[2] := 'off';
   instHMISettings.instAniPNTmr.stations.me[7].kp8Config.colorOn1[3] := 'yellow';
   instHMISettings.instAniPNTmr.stations.me[7].kp8Config.colorOn1[4] := 'off';
   instHMISettings.instAniPNTmr.stations.me[7].kp8Config.colorOn1[5] := 'off';
   instHMISettings.instAniPNTmr.stations.me[7].kp8Config.colorOn1[6] := 'yellow';
   instHMISettings.instAniPNTmr.stations.me[7].kp8Config.colorOn1[7] := 'yellow';
   instHMISettings.instAniPNTmr.stations.me[7].kp8Config.colorOn2[0] := 'off';
   instHMISettings.instAniPNTmr.stations.me[7].kp8Config.colorOn2[1] := 'off';
   instHMISettings.instAniPNTmr.stations.me[7].kp8Config.colorOn2[2] := 'off';
   instHMISettings.instAniPNTmr.stations.me[7].kp8Config.colorOn2[4] := 'off';
   instHMISettings.instAniPNTmr.stations.me[7].kp8Config.colorOn2[5] := 'off';
   instHMISettings.instAniPNTmr.stations.me[7].kp8Config.colorOff[0] := 'off';
   instHMISettings.instAniPNTmr.stations.me[7].kp8Config.colorOff[1] := 'off';
   instHMISettings.instAniPNTmr.stations.me[7].kp8Config.colorOff[2] := 'off';
   instHMISettings.instAniPNTmr.stations.me[7].kp8Config.colorOff[3] := 'green';
   instHMISettings.instAniPNTmr.stations.me[7].kp8Config.colorOff[4] := 'off';
   instHMISettings.instAniPNTmr.stations.me[7].kp8Config.colorOff[5] := 'off';
   instHMISettings.instAniPNTmr.stations.me[7].kp8Config.colorOff[6] := 'green';
   instHMISettings.instAniPNTmr.stations.me[7].kp8Config.colorOff[7] := 'green';
   instHMISettings.instAniPNTmr.stations.me[7].kp8Config.mode[3] := TRUE;
   instHMISettings.instAniPNTmr.stations.me[7].kp8Config.mode[6] := TRUE;
   instHMISettings.instAniPNTmr.stations.me[7].kp8Config.mode[7] := TRUE;
   instHMISettings.instAniPNTmr.stations.me[7].kp8Out := 16#00C8_0000;
   instHMISettings.instAniPNTmr.stations.me[7].line := WSTRING#'VOLVO 16';
   instHMISettings.instAniPNTmr.stations.me[7].partNumbers[0] := WSTRING#'';
   instHMISettings.instAniPNTmr.stations.me[7].partNumbers[1] := WSTRING#'';
   instHMISettings.instAniPNTmr.stations.me[7].partNumbers[2] := WSTRING#'';
   instHMISettings.instAniPNTmr.stations.me[7].partNumbers[3] := WSTRING#'16.32.112.500.520B';
   instHMISettings.instAniPNTmr.stations.me[7].partNumbers[4] := WSTRING#'';
   instHMISettings.instAniPNTmr.stations.me[7].partNumbers[5] := WSTRING#'';
   instHMISettings.instAniPNTmr.stations.me[7].partNumbers[6] := WSTRING#'16.32.112.500.090B';
   instHMISettings.instAniPNTmr.stations.me[7].partNumbers[7] := WSTRING#'16.32.112.500.120A';
   instHMISettings.instAniPNTmr.stations.me[7].presetTime.allotted[3] := 1800.0;
   instHMISettings.instAniPNTmr.stations.me[7].presetTime.allotted[6] := 1800.0;
   instHMISettings.instAniPNTmr.stations.me[7].presetTime.allotted[7] := 1800.0;
   instHMISettings.instAniPNTmr.stations.me[7].presetTime.critical[3] := 300.0;
   instHMISettings.instAniPNTmr.stations.me[7].presetTime.critical[6] := 300.0;
   instHMISettings.instAniPNTmr.stations.me[7].presetTime.critical[7] := 300.0;
   instHMISettings.instAniPNTmr.stations.me[7].settings.btnSelection[3] := TRUE;
   instHMISettings.instAniPNTmr.stations.me[7].stackLightOut := 16#2401_0000;
   instHMISettings.instAniPNTmr.stations.me[8].dropZone := 9;
   instHMISettings.instAniPNTmr.stations.me[8].kp8Config.activate[3] := TRUE;
   instHMISettings.instAniPNTmr.stations.me[8].kp8Config.activate[6] := TRUE;
   instHMISettings.instAniPNTmr.stations.me[8].kp8Config.activate[7] := TRUE;
   instHMISettings.instAniPNTmr.stations.me[8].kp8Config.colorOn1[0] := 'off';
   instHMISettings.instAniPNTmr.stations.me[8].kp8Config.colorOn1[1] := 'off';
   instHMISettings.instAniPNTmr.stations.me[8].kp8Config.colorOn1[2] := 'off';
   instHMISettings.instAniPNTmr.stations.me[8].kp8Config.colorOn1[3] := 'yellow';
   instHMISettings.instAniPNTmr.stations.me[8].kp8Config.colorOn1[4] := 'off';
   instHMISettings.instAniPNTmr.stations.me[8].kp8Config.colorOn1[5] := 'off';
   instHMISettings.instAniPNTmr.stations.me[8].kp8Config.colorOn1[6] := 'yellow';
   instHMISettings.instAniPNTmr.stations.me[8].kp8Config.colorOn1[7] := 'yellow';
   instHMISettings.instAniPNTmr.stations.me[8].kp8Config.colorOn2[0] := 'off';
   instHMISettings.instAniPNTmr.stations.me[8].kp8Config.colorOn2[1] := 'off';
   instHMISettings.instAniPNTmr.stations.me[8].kp8Config.colorOn2[2] := 'off';
   instHMISettings.instAniPNTmr.stations.me[8].kp8Config.colorOn2[4] := 'off';
   instHMISettings.instAniPNTmr.stations.me[8].kp8Config.colorOn2[5] := 'off';
   instHMISettings.instAniPNTmr.stations.me[8].kp8Config.colorOff[0] := 'off';
   instHMISettings.instAniPNTmr.stations.me[8].kp8Config.colorOff[1] := 'off';
   instHMISettings.instAniPNTmr.stations.me[8].kp8Config.colorOff[2] := 'off';
   instHMISettings.instAniPNTmr.stations.me[8].kp8Config.colorOff[3] := 'green';
   instHMISettings.instAniPNTmr.stations.me[8].kp8Config.colorOff[4] := 'off';
   instHMISettings.instAniPNTmr.stations.me[8].kp8Config.colorOff[5] := 'off';
   instHMISettings.instAniPNTmr.stations.me[8].kp8Config.colorOff[6] := 'green';
   instHMISettings.instAniPNTmr.stations.me[8].kp8Config.colorOff[7] := 'green';
   instHMISettings.instAniPNTmr.stations.me[8].kp8Config.mode[3] := TRUE;
   instHMISettings.instAniPNTmr.stations.me[8].kp8Config.mode[6] := TRUE;
   instHMISettings.instAniPNTmr.stations.me[8].kp8Config.mode[7] := TRUE;
   instHMISettings.instAniPNTmr.stations.me[8].kp8Out := 16#00C8_0000;
   instHMISettings.instAniPNTmr.stations.me[8].line := WSTRING#'VOLVO 16';
   instHMISettings.instAniPNTmr.stations.me[8].partNumbers[0] := WSTRING#'';
   instHMISettings.instAniPNTmr.stations.me[8].partNumbers[1] := WSTRING#'';
   instHMISettings.instAniPNTmr.stations.me[8].partNumbers[2] := WSTRING#'';
   instHMISettings.instAniPNTmr.stations.me[8].partNumbers[3] := WSTRING#'16.32.112.580.020A';
   instHMISettings.instAniPNTmr.stations.me[8].partNumbers[4] := WSTRING#'';
   instHMISettings.instAniPNTmr.stations.me[8].partNumbers[5] := WSTRING#'';
   instHMISettings.instAniPNTmr.stations.me[8].partNumbers[6] := WSTRING#'16.32.112.500.300E';
   instHMISettings.instAniPNTmr.stations.me[8].partNumbers[7] := WSTRING#'16.32.112.520.300E';
   instHMISettings.instAniPNTmr.stations.me[8].presetTime.allotted[3] := 1800.0;
   instHMISettings.instAniPNTmr.stations.me[8].presetTime.allotted[6] := 1800.0;
   instHMISettings.instAniPNTmr.stations.me[8].presetTime.allotted[7] := 1800.0;
   instHMISettings.instAniPNTmr.stations.me[8].presetTime.critical[3] := 300.0;
   instHMISettings.instAniPNTmr.stations.me[8].presetTime.critical[6] := 300.0;
   instHMISettings.instAniPNTmr.stations.me[8].presetTime.critical[7] := 300.0;
   instHMISettings.instAniPNTmr.stations.me[8].stackLightOut := 16#2401_0000;
   instHMISettings.instAniPNTmr.stations.me[9].dropZone := 10;
   instHMISettings.instAniPNTmr.stations.me[9].kp8Config.activate[3] := TRUE;
   instHMISettings.instAniPNTmr.stations.me[9].kp8Config.activate[7] := TRUE;
   instHMISettings.instAniPNTmr.stations.me[9].kp8Config.colorOn1[0] := 'off';
   instHMISettings.instAniPNTmr.stations.me[9].kp8Config.colorOn1[1] := 'off';
   instHMISettings.instAniPNTmr.stations.me[9].kp8Config.colorOn1[2] := 'off';
   instHMISettings.instAniPNTmr.stations.me[9].kp8Config.colorOn1[3] := 'yellow';
   instHMISettings.instAniPNTmr.stations.me[9].kp8Config.colorOn1[4] := 'off';
   instHMISettings.instAniPNTmr.stations.me[9].kp8Config.colorOn1[5] := 'off';
   instHMISettings.instAniPNTmr.stations.me[9].kp8Config.colorOn1[6] := 'off';
   instHMISettings.instAniPNTmr.stations.me[9].kp8Config.colorOn1[7] := 'yellow';
   instHMISettings.instAniPNTmr.stations.me[9].kp8Config.colorOn2[0] := 'off';
   instHMISettings.instAniPNTmr.stations.me[9].kp8Config.colorOn2[1] := 'off';
   instHMISettings.instAniPNTmr.stations.me[9].kp8Config.colorOn2[2] := 'off';
   instHMISettings.instAniPNTmr.stations.me[9].kp8Config.colorOn2[4] := 'off';
   instHMISettings.instAniPNTmr.stations.me[9].kp8Config.colorOn2[5] := 'off';
   instHMISettings.instAniPNTmr.stations.me[9].kp8Config.colorOn2[6] := 'off';
   instHMISettings.instAniPNTmr.stations.me[9].kp8Config.colorOff[0] := 'off';
   instHMISettings.instAniPNTmr.stations.me[9].kp8Config.colorOff[1] := 'off';
   instHMISettings.instAniPNTmr.stations.me[9].kp8Config.colorOff[2] := 'off';
   instHMISettings.instAniPNTmr.stations.me[9].kp8Config.colorOff[3] := 'green';
   instHMISettings.instAniPNTmr.stations.me[9].kp8Config.colorOff[4] := 'off';
   instHMISettings.instAniPNTmr.stations.me[9].kp8Config.colorOff[5] := 'off';
   instHMISettings.instAniPNTmr.stations.me[9].kp8Config.colorOff[6] := 'off';
   instHMISettings.instAniPNTmr.stations.me[9].kp8Config.colorOff[7] := 'green';
   instHMISettings.instAniPNTmr.stations.me[9].kp8Config.mode[3] := TRUE;
   instHMISettings.instAniPNTmr.stations.me[9].kp8Config.mode[7] := TRUE;
   instHMISettings.instAniPNTmr.stations.me[9].kp8Out := 16#0088_0000;
   instHMISettings.instAniPNTmr.stations.me[9].line := WSTRING#'VOLVO 16';
   instHMISettings.instAniPNTmr.stations.me[9].partNumbers[0] := WSTRING#'';
   instHMISettings.instAniPNTmr.stations.me[9].partNumbers[1] := WSTRING#'';
   instHMISettings.instAniPNTmr.stations.me[9].partNumbers[2] := WSTRING#'';
   instHMISettings.instAniPNTmr.stations.me[9].partNumbers[3] := WSTRING#'16.32.112.757.001A';
   instHMISettings.instAniPNTmr.stations.me[9].partNumbers[4] := WSTRING#'';
   instHMISettings.instAniPNTmr.stations.me[9].partNumbers[5] := WSTRING#'';
   instHMISettings.instAniPNTmr.stations.me[9].partNumbers[6] := WSTRING#'';
   instHMISettings.instAniPNTmr.stations.me[9].partNumbers[7] := WSTRING#'16.32.112.757.000A';
   instHMISettings.instAniPNTmr.stations.me[9].presetTime.allotted[3] := 1800.0;
   instHMISettings.instAniPNTmr.stations.me[9].presetTime.allotted[7] := 1800.0;
   instHMISettings.instAniPNTmr.stations.me[9].presetTime.critical[3] := 300.0;
   instHMISettings.instAniPNTmr.stations.me[9].presetTime.critical[7] := 300.0;
   instHMISettings.instAniPNTmr.stations.me[9].stackLightOut := 16#2400_0000;
   instHMISettings.instAniPNTmr.stations.me[10].dropZone := 11;
   instHMISettings.instAniPNTmr.stations.me[10].kp8Config.activate[3] := TRUE;
   instHMISettings.instAniPNTmr.stations.me[10].kp8Config.activate[6] := TRUE;
   instHMISettings.instAniPNTmr.stations.me[10].kp8Config.activate[7] := TRUE;
   instHMISettings.instAniPNTmr.stations.me[10].kp8Config.colorOn1[0] := 'off';
   instHMISettings.instAniPNTmr.stations.me[10].kp8Config.colorOn1[1] := 'off';
   instHMISettings.instAniPNTmr.stations.me[10].kp8Config.colorOn1[2] := 'off';
   instHMISettings.instAniPNTmr.stations.me[10].kp8Config.colorOn1[3] := 'yellow';
   instHMISettings.instAniPNTmr.stations.me[10].kp8Config.colorOn1[4] := 'off';
   instHMISettings.instAniPNTmr.stations.me[10].kp8Config.colorOn1[5] := 'off';
   instHMISettings.instAniPNTmr.stations.me[10].kp8Config.colorOn1[6] := 'yellow';
   instHMISettings.instAniPNTmr.stations.me[10].kp8Config.colorOn1[7] := 'yellow';
   instHMISettings.instAniPNTmr.stations.me[10].kp8Config.colorOn2[0] := 'off';
   instHMISettings.instAniPNTmr.stations.me[10].kp8Config.colorOn2[1] := 'off';
   instHMISettings.instAniPNTmr.stations.me[10].kp8Config.colorOn2[2] := 'off';
   instHMISettings.instAniPNTmr.stations.me[10].kp8Config.colorOn2[4] := 'off';
   instHMISettings.instAniPNTmr.stations.me[10].kp8Config.colorOn2[5] := 'off';
   instHMISettings.instAniPNTmr.stations.me[10].kp8Config.colorOff[0] := 'off';
   instHMISettings.instAniPNTmr.stations.me[10].kp8Config.colorOff[1] := 'off';
   instHMISettings.instAniPNTmr.stations.me[10].kp8Config.colorOff[2] := 'off';
   instHMISettings.instAniPNTmr.stations.me[10].kp8Config.colorOff[3] := 'green';
   instHMISettings.instAniPNTmr.stations.me[10].kp8Config.colorOff[4] := 'off';
   instHMISettings.instAniPNTmr.stations.me[10].kp8Config.colorOff[5] := 'off';
   instHMISettings.instAniPNTmr.stations.me[10].kp8Config.colorOff[6] := 'green';
   instHMISettings.instAniPNTmr.stations.me[10].kp8Config.colorOff[7] := 'green';
   instHMISettings.instAniPNTmr.stations.me[10].kp8Config.mode[3] := TRUE;
   instHMISettings.instAniPNTmr.stations.me[10].kp8Config.mode[6] := TRUE;
   instHMISettings.instAniPNTmr.stations.me[10].kp8Config.mode[7] := TRUE;
   instHMISettings.instAniPNTmr.stations.me[10].kp8Out := 16#00C8_0000;
   instHMISettings.instAniPNTmr.stations.me[10].line := WSTRING#'VOLVO 16';
   instHMISettings.instAniPNTmr.stations.me[10].partNumbers[0] := WSTRING#'';
   instHMISettings.instAniPNTmr.stations.me[10].partNumbers[1] := WSTRING#'';
   instHMISettings.instAniPNTmr.stations.me[10].partNumbers[2] := WSTRING#'';
   instHMISettings.instAniPNTmr.stations.me[10].partNumbers[3] := WSTRING#'16.32.112.500.150B';
   instHMISettings.instAniPNTmr.stations.me[10].partNumbers[4] := WSTRING#'';
   instHMISettings.instAniPNTmr.stations.me[10].partNumbers[5] := WSTRING#'';
   instHMISettings.instAniPNTmr.stations.me[10].partNumbers[6] := WSTRING#'16.32.806.502.080A';
   instHMISettings.instAniPNTmr.stations.me[10].partNumbers[7] := WSTRING#'16.32.112.500.160A';
   instHMISettings.instAniPNTmr.stations.me[10].presetTime.allotted[3] := 1800.0;
   instHMISettings.instAniPNTmr.stations.me[10].presetTime.allotted[6] := 1800.0;
   instHMISettings.instAniPNTmr.stations.me[10].presetTime.allotted[7] := 1800.0;
   instHMISettings.instAniPNTmr.stations.me[10].presetTime.critical[3] := 300.0;
   instHMISettings.instAniPNTmr.stations.me[10].presetTime.critical[6] := 300.0;
   instHMISettings.instAniPNTmr.stations.me[10].presetTime.critical[7] := 300.0;
   instHMISettings.instAniPNTmr.stations.me[10].stackLightOut := 16#2401_0000;
   instHMISettings.instAniPNTmr.stations.me[11].dropZone := 1;
   instHMISettings.instAniPNTmr.stations.me[11].kp8Config.activate[3] := TRUE;
   instHMISettings.instAniPNTmr.stations.me[11].kp8Config.activate[6] := TRUE;
   instHMISettings.instAniPNTmr.stations.me[11].kp8Config.activate[7] := TRUE;
   instHMISettings.instAniPNTmr.stations.me[11].kp8Config.colorOn1[0] := 'off';
   instHMISettings.instAniPNTmr.stations.me[11].kp8Config.colorOn1[1] := 'off';
   instHMISettings.instAniPNTmr.stations.me[11].kp8Config.colorOn1[2] := 'off';
   instHMISettings.instAniPNTmr.stations.me[11].kp8Config.colorOn1[3] := 'yellow';
   instHMISettings.instAniPNTmr.stations.me[11].kp8Config.colorOn1[4] := 'off';
   instHMISettings.instAniPNTmr.stations.me[11].kp8Config.colorOn1[5] := 'off';
   instHMISettings.instAniPNTmr.stations.me[11].kp8Config.colorOn1[6] := 'yellow';
   instHMISettings.instAniPNTmr.stations.me[11].kp8Config.colorOn1[7] := 'yellow';
   instHMISettings.instAniPNTmr.stations.me[11].kp8Config.colorOn2[0] := 'off';
   instHMISettings.instAniPNTmr.stations.me[11].kp8Config.colorOn2[1] := 'off';
   instHMISettings.instAniPNTmr.stations.me[11].kp8Config.colorOn2[2] := 'off';
   instHMISettings.instAniPNTmr.stations.me[11].kp8Config.colorOn2[4] := 'off';
   instHMISettings.instAniPNTmr.stations.me[11].kp8Config.colorOn2[5] := 'off';
   instHMISettings.instAniPNTmr.stations.me[11].kp8Config.colorOff[0] := 'off';
   instHMISettings.instAniPNTmr.stations.me[11].kp8Config.colorOff[1] := 'off';
   instHMISettings.instAniPNTmr.stations.me[11].kp8Config.colorOff[2] := 'off';
   instHMISettings.instAniPNTmr.stations.me[11].kp8Config.colorOff[3] := 'green';
   instHMISettings.instAniPNTmr.stations.me[11].kp8Config.colorOff[4] := 'off';
   instHMISettings.instAniPNTmr.stations.me[11].kp8Config.colorOff[5] := 'off';
   instHMISettings.instAniPNTmr.stations.me[11].kp8Config.colorOff[6] := 'green';
   instHMISettings.instAniPNTmr.stations.me[11].kp8Config.colorOff[7] := 'green';
   instHMISettings.instAniPNTmr.stations.me[11].kp8Config.mode[3] := TRUE;
   instHMISettings.instAniPNTmr.stations.me[11].kp8Config.mode[6] := TRUE;
   instHMISettings.instAniPNTmr.stations.me[11].kp8Config.mode[7] := TRUE;
   instHMISettings.instAniPNTmr.stations.me[11].kp8Out := 16#00C8_0000;
   instHMISettings.instAniPNTmr.stations.me[11].line := WSTRING#'CHM';
   instHMISettings.instAniPNTmr.stations.me[11].partNumbers[0] := WSTRING#'';
   instHMISettings.instAniPNTmr.stations.me[11].partNumbers[1] := WSTRING#'';
   instHMISettings.instAniPNTmr.stations.me[11].partNumbers[2] := WSTRING#'';
   instHMISettings.instAniPNTmr.stations.me[11].partNumbers[3] := WSTRING#'16.08.216.515.008C';
   instHMISettings.instAniPNTmr.stations.me[11].partNumbers[4] := WSTRING#'';
   instHMISettings.instAniPNTmr.stations.me[11].partNumbers[5] := WSTRING#'';
   instHMISettings.instAniPNTmr.stations.me[11].partNumbers[6] := WSTRING#'16.08.216.181.110B';
   instHMISettings.instAniPNTmr.stations.me[11].partNumbers[7] := WSTRING#'16.08.208.131.010L';
   instHMISettings.instAniPNTmr.stations.me[11].presetTime.allotted[3] := 1800.0;
   instHMISettings.instAniPNTmr.stations.me[11].presetTime.allotted[6] := 1800.0;
   instHMISettings.instAniPNTmr.stations.me[11].presetTime.allotted[7] := 1800.0;
   instHMISettings.instAniPNTmr.stations.me[11].presetTime.critical[3] := 300.0;
   instHMISettings.instAniPNTmr.stations.me[11].presetTime.critical[6] := 300.0;
   instHMISettings.instAniPNTmr.stations.me[11].presetTime.critical[7] := 300.0;
   instHMISettings.instAniPNTmr.stations.me[11].stackLightOut := 16#2401_0000;
   instHMISettings.instAniPNTmr.stations.me[12].dropZone := 2;
   instHMISettings.instAniPNTmr.stations.me[12].kp8Config.activate[1] := TRUE;
   instHMISettings.instAniPNTmr.stations.me[12].kp8Config.activate[2] := TRUE;
   instHMISettings.instAniPNTmr.stations.me[12].kp8Config.activate[3] := TRUE;
   instHMISettings.instAniPNTmr.stations.me[12].kp8Config.activate[5] := TRUE;
   instHMISettings.instAniPNTmr.stations.me[12].kp8Config.activate[6] := TRUE;
   instHMISettings.instAniPNTmr.stations.me[12].kp8Config.activate[7] := TRUE;
   instHMISettings.instAniPNTmr.stations.me[12].kp8Config.colorOn1[0] := 'off';
   instHMISettings.instAniPNTmr.stations.me[12].kp8Config.colorOn1[1] := 'yellow';
   instHMISettings.instAniPNTmr.stations.me[12].kp8Config.colorOn1[2] := 'yellow';
   instHMISettings.instAniPNTmr.stations.me[12].kp8Config.colorOn1[3] := 'yellow';
   instHMISettings.instAniPNTmr.stations.me[12].kp8Config.colorOn1[4] := 'off';
   instHMISettings.instAniPNTmr.stations.me[12].kp8Config.colorOn1[5] := 'yellow';
   instHMISettings.instAniPNTmr.stations.me[12].kp8Config.colorOn1[6] := 'yellow';
   instHMISettings.instAniPNTmr.stations.me[12].kp8Config.colorOn1[7] := 'yellow';
   instHMISettings.instAniPNTmr.stations.me[12].kp8Config.colorOn2[0] := 'off';
   instHMISettings.instAniPNTmr.stations.me[12].kp8Config.colorOn2[4] := 'off';
   instHMISettings.instAniPNTmr.stations.me[12].kp8Config.colorOff[0] := 'off';
   instHMISettings.instAniPNTmr.stations.me[12].kp8Config.colorOff[1] := 'green';
   instHMISettings.instAniPNTmr.stations.me[12].kp8Config.colorOff[2] := 'green';
   instHMISettings.instAniPNTmr.stations.me[12].kp8Config.colorOff[3] := 'green';
   instHMISettings.instAniPNTmr.stations.me[12].kp8Config.colorOff[4] := 'off';
   instHMISettings.instAniPNTmr.stations.me[12].kp8Config.colorOff[5] := 'green';
   instHMISettings.instAniPNTmr.stations.me[12].kp8Config.colorOff[6] := 'green';
   instHMISettings.instAniPNTmr.stations.me[12].kp8Config.colorOff[7] := 'green';
   instHMISettings.instAniPNTmr.stations.me[12].kp8Config.mode[1] := TRUE;
   instHMISettings.instAniPNTmr.stations.me[12].kp8Config.mode[2] := TRUE;
   instHMISettings.instAniPNTmr.stations.me[12].kp8Config.mode[3] := TRUE;
   instHMISettings.instAniPNTmr.stations.me[12].kp8Config.mode[5] := TRUE;
   instHMISettings.instAniPNTmr.stations.me[12].kp8Config.mode[6] := TRUE;
   instHMISettings.instAniPNTmr.stations.me[12].kp8Config.mode[7] := TRUE;
   instHMISettings.instAniPNTmr.stations.me[12].kp8Out := 16#00EE_0000;
   instHMISettings.instAniPNTmr.stations.me[12].line := WSTRING#'CHM';
   instHMISettings.instAniPNTmr.stations.me[12].partNumbers[0] := WSTRING#'';
   instHMISettings.instAniPNTmr.stations.me[12].partNumbers[1] := WSTRING#'16.08.216.526.009B';
   instHMISettings.instAniPNTmr.stations.me[12].partNumbers[2] := WSTRING#'16.08.216.871.010C';
   instHMISettings.instAniPNTmr.stations.me[12].partNumbers[3] := WSTRING#'16.08.216.141.010C';
   instHMISettings.instAniPNTmr.stations.me[12].partNumbers[4] := WSTRING#'';
   instHMISettings.instAniPNTmr.stations.me[12].partNumbers[5] := WSTRING#'16.08.216.526.002D';
   instHMISettings.instAniPNTmr.stations.me[12].partNumbers[6] := WSTRING#'16.08.215.871.010C';
   instHMISettings.instAniPNTmr.stations.me[12].partNumbers[7] := WSTRING#'16.08.215.141.010C';
   instHMISettings.instAniPNTmr.stations.me[12].presetTime.allotted[1] := 1800.0;
   instHMISettings.instAniPNTmr.stations.me[12].presetTime.allotted[2] := 1800.0;
   instHMISettings.instAniPNTmr.stations.me[12].presetTime.allotted[3] := 1800.0;
   instHMISettings.instAniPNTmr.stations.me[12].presetTime.allotted[5] := 1800.0;
   instHMISettings.instAniPNTmr.stations.me[12].presetTime.allotted[6] := 1800.0;
   instHMISettings.instAniPNTmr.stations.me[12].presetTime.allotted[7] := 1800.0;
   instHMISettings.instAniPNTmr.stations.me[12].presetTime.critical[1] := 300.0;
   instHMISettings.instAniPNTmr.stations.me[12].presetTime.critical[2] := 300.0;
   instHMISettings.instAniPNTmr.stations.me[12].presetTime.critical[3] := 300.0;
   instHMISettings.instAniPNTmr.stations.me[12].presetTime.critical[5] := 300.0;
   instHMISettings.instAniPNTmr.stations.me[12].presetTime.critical[6] := 300.0;
   instHMISettings.instAniPNTmr.stations.me[12].presetTime.critical[7] := 300.0;
   instHMISettings.instAniPNTmr.stations.me[12].stackLightOut := 16#2449_0200;
   instHMISettings.instAniPNTmr.stations.me[13].dropZone := 3;
   instHMISettings.instAniPNTmr.stations.me[13].kp8Config.activate[2] := TRUE;
   instHMISettings.instAniPNTmr.stations.me[13].kp8Config.activate[3] := TRUE;
   instHMISettings.instAniPNTmr.stations.me[13].kp8Config.activate[6] := TRUE;
   instHMISettings.instAniPNTmr.stations.me[13].kp8Config.activate[7] := TRUE;
   instHMISettings.instAniPNTmr.stations.me[13].kp8Config.colorOn1[0] := 'off';
   instHMISettings.instAniPNTmr.stations.me[13].kp8Config.colorOn1[1] := 'off';
   instHMISettings.instAniPNTmr.stations.me[13].kp8Config.colorOn1[2] := 'yellow';
   instHMISettings.instAniPNTmr.stations.me[13].kp8Config.colorOn1[3] := 'yellow';
   instHMISettings.instAniPNTmr.stations.me[13].kp8Config.colorOn1[4] := 'off';
   instHMISettings.instAniPNTmr.stations.me[13].kp8Config.colorOn1[5] := 'off';
   instHMISettings.instAniPNTmr.stations.me[13].kp8Config.colorOn1[6] := 'yellow';
   instHMISettings.instAniPNTmr.stations.me[13].kp8Config.colorOn1[7] := 'yellow';
   instHMISettings.instAniPNTmr.stations.me[13].kp8Config.colorOn2[0] := 'off';
   instHMISettings.instAniPNTmr.stations.me[13].kp8Config.colorOn2[1] := 'off';
   instHMISettings.instAniPNTmr.stations.me[13].kp8Config.colorOn2[4] := 'off';
   instHMISettings.instAniPNTmr.stations.me[13].kp8Config.colorOn2[5] := 'off';
   instHMISettings.instAniPNTmr.stations.me[13].kp8Config.colorOff[0] := 'off';
   instHMISettings.instAniPNTmr.stations.me[13].kp8Config.colorOff[1] := 'off';
   instHMISettings.instAniPNTmr.stations.me[13].kp8Config.colorOff[2] := 'green';
   instHMISettings.instAniPNTmr.stations.me[13].kp8Config.colorOff[3] := 'green';
   instHMISettings.instAniPNTmr.stations.me[13].kp8Config.colorOff[4] := 'off';
   instHMISettings.instAniPNTmr.stations.me[13].kp8Config.colorOff[5] := 'off';
   instHMISettings.instAniPNTmr.stations.me[13].kp8Config.colorOff[6] := 'green';
   instHMISettings.instAniPNTmr.stations.me[13].kp8Config.colorOff[7] := 'green';
   instHMISettings.instAniPNTmr.stations.me[13].kp8Config.mode[2] := TRUE;
   instHMISettings.instAniPNTmr.stations.me[13].kp8Config.mode[3] := TRUE;
   instHMISettings.instAniPNTmr.stations.me[13].kp8Config.mode[6] := TRUE;
   instHMISettings.instAniPNTmr.stations.me[13].kp8Config.mode[7] := TRUE;
   instHMISettings.instAniPNTmr.stations.me[13].kp8Out := 16#00CC_0000;
   instHMISettings.instAniPNTmr.stations.me[13].line := WSTRING#'CHM';
   instHMISettings.instAniPNTmr.stations.me[13].partNumbers[0] := WSTRING#'';
   instHMISettings.instAniPNTmr.stations.me[13].partNumbers[1] := WSTRING#'';
   instHMISettings.instAniPNTmr.stations.me[13].partNumbers[2] := WSTRING#'16.08.216.251.000B';
   instHMISettings.instAniPNTmr.stations.me[13].partNumbers[3] := WSTRING#'16.08.208.901.000G';
   instHMISettings.instAniPNTmr.stations.me[13].partNumbers[4] := WSTRING#'';
   instHMISettings.instAniPNTmr.stations.me[13].partNumbers[5] := WSTRING#'';
   instHMISettings.instAniPNTmr.stations.me[13].partNumbers[6] := WSTRING#'16.08.208.911.000H';
   instHMISettings.instAniPNTmr.stations.me[13].partNumbers[7] := WSTRING#'16.08.216.911.000C';
   instHMISettings.instAniPNTmr.stations.me[13].presetTime.allotted[2] := 1800.0;
   instHMISettings.instAniPNTmr.stations.me[13].presetTime.allotted[3] := 1800.0;
   instHMISettings.instAniPNTmr.stations.me[13].presetTime.allotted[6] := 1800.0;
   instHMISettings.instAniPNTmr.stations.me[13].presetTime.allotted[7] := 1800.0;
   instHMISettings.instAniPNTmr.stations.me[13].presetTime.critical[2] := 300.0;
   instHMISettings.instAniPNTmr.stations.me[13].presetTime.critical[3] := 300.0;
   instHMISettings.instAniPNTmr.stations.me[13].presetTime.critical[6] := 300.0;
   instHMISettings.instAniPNTmr.stations.me[13].presetTime.critical[7] := 300.0;
   instHMISettings.instAniPNTmr.stations.me[13].stackLightOut := 16#2409_0000;
   instHMISettings.instAniPNTmr.stations.me[14].dropZone := 4;
   instHMISettings.instAniPNTmr.stations.me[14].kp8Config.activate[2] := TRUE;
   instHMISettings.instAniPNTmr.stations.me[14].kp8Config.activate[3] := TRUE;
   instHMISettings.instAniPNTmr.stations.me[14].kp8Config.activate[5] := TRUE;
   instHMISettings.instAniPNTmr.stations.me[14].kp8Config.activate[6] := TRUE;
   instHMISettings.instAniPNTmr.stations.me[14].kp8Config.activate[7] := TRUE;
   instHMISettings.instAniPNTmr.stations.me[14].kp8Config.colorOn1[0] := 'off';
   instHMISettings.instAniPNTmr.stations.me[14].kp8Config.colorOn1[1] := 'off';
   instHMISettings.instAniPNTmr.stations.me[14].kp8Config.colorOn1[2] := 'yellow';
   instHMISettings.instAniPNTmr.stations.me[14].kp8Config.colorOn1[3] := 'yellow';
   instHMISettings.instAniPNTmr.stations.me[14].kp8Config.colorOn1[4] := 'off';
   instHMISettings.instAniPNTmr.stations.me[14].kp8Config.colorOn1[5] := 'yellow';
   instHMISettings.instAniPNTmr.stations.me[14].kp8Config.colorOn1[6] := 'yellow';
   instHMISettings.instAniPNTmr.stations.me[14].kp8Config.colorOn1[7] := 'yellow';
   instHMISettings.instAniPNTmr.stations.me[14].kp8Config.colorOn2[0] := 'off';
   instHMISettings.instAniPNTmr.stations.me[14].kp8Config.colorOn2[1] := 'off';
   instHMISettings.instAniPNTmr.stations.me[14].kp8Config.colorOn2[4] := 'off';
   instHMISettings.instAniPNTmr.stations.me[14].kp8Config.colorOff[0] := 'off';
   instHMISettings.instAniPNTmr.stations.me[14].kp8Config.colorOff[1] := 'off';
   instHMISettings.instAniPNTmr.stations.me[14].kp8Config.colorOff[2] := 'green';
   instHMISettings.instAniPNTmr.stations.me[14].kp8Config.colorOff[3] := 'green';
   instHMISettings.instAniPNTmr.stations.me[14].kp8Config.colorOff[4] := 'off';
   instHMISettings.instAniPNTmr.stations.me[14].kp8Config.colorOff[5] := 'green';
   instHMISettings.instAniPNTmr.stations.me[14].kp8Config.colorOff[6] := 'green';
   instHMISettings.instAniPNTmr.stations.me[14].kp8Config.colorOff[7] := 'green';
   instHMISettings.instAniPNTmr.stations.me[14].kp8Config.mode[2] := TRUE;
   instHMISettings.instAniPNTmr.stations.me[14].kp8Config.mode[3] := TRUE;
   instHMISettings.instAniPNTmr.stations.me[14].kp8Config.mode[5] := TRUE;
   instHMISettings.instAniPNTmr.stations.me[14].kp8Config.mode[6] := TRUE;
   instHMISettings.instAniPNTmr.stations.me[14].kp8Config.mode[7] := TRUE;
   instHMISettings.instAniPNTmr.stations.me[14].kp8Out := 16#00EC_0000;
   instHMISettings.instAniPNTmr.stations.me[14].line := WSTRING#'CHM';
   instHMISettings.instAniPNTmr.stations.me[14].partNumbers[0] := WSTRING#'';
   instHMISettings.instAniPNTmr.stations.me[14].partNumbers[1] := WSTRING#'';
   instHMISettings.instAniPNTmr.stations.me[14].partNumbers[2] := WSTRING#'16.08.216.181.100A';
   instHMISettings.instAniPNTmr.stations.me[14].partNumbers[3] := WSTRING#'16.08.216.910.020B';
   instHMISettings.instAniPNTmr.stations.me[14].partNumbers[4] := WSTRING#'';
   instHMISettings.instAniPNTmr.stations.me[14].partNumbers[5] := WSTRING#'16.08.216.181.090A';
   instHMISettings.instAniPNTmr.stations.me[14].partNumbers[6] := WSTRING#'16.08.216.722.001A';
   instHMISettings.instAniPNTmr.stations.me[14].partNumbers[7] := WSTRING#'16.08.216.181.010B';
   instHMISettings.instAniPNTmr.stations.me[14].presetTime.allotted[2] := 1800.0;
   instHMISettings.instAniPNTmr.stations.me[14].presetTime.allotted[3] := 1800.0;
   instHMISettings.instAniPNTmr.stations.me[14].presetTime.allotted[5] := 1800.0;
   instHMISettings.instAniPNTmr.stations.me[14].presetTime.allotted[6] := 1800.0;
   instHMISettings.instAniPNTmr.stations.me[14].presetTime.allotted[7] := 1800.0;
   instHMISettings.instAniPNTmr.stations.me[14].presetTime.critical[2] := 300.0;
   instHMISettings.instAniPNTmr.stations.me[14].presetTime.critical[3] := 300.0;
   instHMISettings.instAniPNTmr.stations.me[14].presetTime.critical[5] := 300.0;
   instHMISettings.instAniPNTmr.stations.me[14].presetTime.critical[6] := 300.0;
   instHMISettings.instAniPNTmr.stations.me[14].presetTime.critical[7] := 300.0;
   instHMISettings.instAniPNTmr.stations.me[14].stackLightOut := 16#2449_0000;
   instHMISettings.instAniPNTmr.stations.me[15].dropZone := 5;
   instHMISettings.instAniPNTmr.stations.me[15].kp8Config.activate[1] := TRUE;
   instHMISettings.instAniPNTmr.stations.me[15].kp8Config.activate[2] := TRUE;
   instHMISettings.instAniPNTmr.stations.me[15].kp8Config.activate[3] := TRUE;
   instHMISettings.instAniPNTmr.stations.me[15].kp8Config.activate[5] := TRUE;
   instHMISettings.instAniPNTmr.stations.me[15].kp8Config.activate[6] := TRUE;
   instHMISettings.instAniPNTmr.stations.me[15].kp8Config.activate[7] := TRUE;
   instHMISettings.instAniPNTmr.stations.me[15].kp8Config.colorOn1[0] := 'off';
   instHMISettings.instAniPNTmr.stations.me[15].kp8Config.colorOn1[1] := 'yellow';
   instHMISettings.instAniPNTmr.stations.me[15].kp8Config.colorOn1[2] := 'yellow';
   instHMISettings.instAniPNTmr.stations.me[15].kp8Config.colorOn1[3] := 'yellow';
   instHMISettings.instAniPNTmr.stations.me[15].kp8Config.colorOn1[4] := 'off';
   instHMISettings.instAniPNTmr.stations.me[15].kp8Config.colorOn1[5] := 'yellow';
   instHMISettings.instAniPNTmr.stations.me[15].kp8Config.colorOn1[6] := 'yellow';
   instHMISettings.instAniPNTmr.stations.me[15].kp8Config.colorOn1[7] := 'yellow';
   instHMISettings.instAniPNTmr.stations.me[15].kp8Config.colorOn2[0] := 'off';
   instHMISettings.instAniPNTmr.stations.me[15].kp8Config.colorOn2[4] := 'off';
   instHMISettings.instAniPNTmr.stations.me[15].kp8Config.colorOff[0] := 'off';
   instHMISettings.instAniPNTmr.stations.me[15].kp8Config.colorOff[1] := 'green';
   instHMISettings.instAniPNTmr.stations.me[15].kp8Config.colorOff[2] := 'green';
   instHMISettings.instAniPNTmr.stations.me[15].kp8Config.colorOff[3] := 'green';
   instHMISettings.instAniPNTmr.stations.me[15].kp8Config.colorOff[4] := 'off';
   instHMISettings.instAniPNTmr.stations.me[15].kp8Config.colorOff[5] := 'green';
   instHMISettings.instAniPNTmr.stations.me[15].kp8Config.colorOff[6] := 'green';
   instHMISettings.instAniPNTmr.stations.me[15].kp8Config.colorOff[7] := 'green';
   instHMISettings.instAniPNTmr.stations.me[15].kp8Config.mode[1] := TRUE;
   instHMISettings.instAniPNTmr.stations.me[15].kp8Config.mode[2] := TRUE;
   instHMISettings.instAniPNTmr.stations.me[15].kp8Config.mode[3] := TRUE;
   instHMISettings.instAniPNTmr.stations.me[15].kp8Config.mode[5] := TRUE;
   instHMISettings.instAniPNTmr.stations.me[15].kp8Config.mode[6] := TRUE;
   instHMISettings.instAniPNTmr.stations.me[15].kp8Config.mode[7] := TRUE;
   instHMISettings.instAniPNTmr.stations.me[15].kp8Out := 16#00EE_0000;
   instHMISettings.instAniPNTmr.stations.me[15].line := WSTRING#'CHM';
   instHMISettings.instAniPNTmr.stations.me[15].partNumbers[0] := WSTRING#'';
   instHMISettings.instAniPNTmr.stations.me[15].partNumbers[1] := WSTRING#'16.08.211.551.000B';
   instHMISettings.instAniPNTmr.stations.me[15].partNumbers[2] := WSTRING#'16.08.216.511.000C';
   instHMISettings.instAniPNTmr.stations.me[15].partNumbers[3] := WSTRING#'16.08.208.501.000B';
   instHMISettings.instAniPNTmr.stations.me[15].partNumbers[4] := WSTRING#'';
   instHMISettings.instAniPNTmr.stations.me[15].partNumbers[5] := WSTRING#'16.08.216.551.000B';
   instHMISettings.instAniPNTmr.stations.me[15].partNumbers[6] := WSTRING#'16.08.216.231.000B';
   instHMISettings.instAniPNTmr.stations.me[15].partNumbers[7] := WSTRING#'16.08.216.501.000C';
   instHMISettings.instAniPNTmr.stations.me[15].presetTime.allotted[1] := 1800.0;
   instHMISettings.instAniPNTmr.stations.me[15].presetTime.allotted[2] := 1800.0;
   instHMISettings.instAniPNTmr.stations.me[15].presetTime.allotted[3] := 1800.0;
   instHMISettings.instAniPNTmr.stations.me[15].presetTime.allotted[5] := 1800.0;
   instHMISettings.instAniPNTmr.stations.me[15].presetTime.allotted[6] := 1800.0;
   instHMISettings.instAniPNTmr.stations.me[15].presetTime.allotted[7] := 1800.0;
   instHMISettings.instAniPNTmr.stations.me[15].presetTime.critical[1] := 300.0;
   instHMISettings.instAniPNTmr.stations.me[15].presetTime.critical[2] := 300.0;
   instHMISettings.instAniPNTmr.stations.me[15].presetTime.critical[3] := 300.0;
   instHMISettings.instAniPNTmr.stations.me[15].presetTime.critical[5] := 300.0;
   instHMISettings.instAniPNTmr.stations.me[15].presetTime.critical[6] := 300.0;
   instHMISettings.instAniPNTmr.stations.me[15].presetTime.critical[7] := 300.0;
   instHMISettings.instAniPNTmr.stations.me[15].stackLightOut := 16#2449_0200;
   instHMISettings.instAniPNTmr.stations.me[16].dropZone := 1;
   instHMISettings.instAniPNTmr.stations.me[16].kp8Config.activate[3] := TRUE;
   instHMISettings.instAniPNTmr.stations.me[16].kp8Config.activate[7] := TRUE;
   instHMISettings.instAniPNTmr.stations.me[16].kp8Config.colorOn1[0] := 'off';
   instHMISettings.instAniPNTmr.stations.me[16].kp8Config.colorOn1[1] := 'off';
   instHMISettings.instAniPNTmr.stations.me[16].kp8Config.colorOn1[2] := 'off';
   instHMISettings.instAniPNTmr.stations.me[16].kp8Config.colorOn1[3] := 'yellow';
   instHMISettings.instAniPNTmr.stations.me[16].kp8Config.colorOn1[4] := 'off';
   instHMISettings.instAniPNTmr.stations.me[16].kp8Config.colorOn1[5] := 'off';
   instHMISettings.instAniPNTmr.stations.me[16].kp8Config.colorOn1[6] := 'off';
   instHMISettings.instAniPNTmr.stations.me[16].kp8Config.colorOn1[7] := 'yellow';
   instHMISettings.instAniPNTmr.stations.me[16].kp8Config.colorOn2[0] := 'off';
   instHMISettings.instAniPNTmr.stations.me[16].kp8Config.colorOn2[1] := 'off';
   instHMISettings.instAniPNTmr.stations.me[16].kp8Config.colorOn2[2] := 'off';
   instHMISettings.instAniPNTmr.stations.me[16].kp8Config.colorOn2[4] := 'off';
   instHMISettings.instAniPNTmr.stations.me[16].kp8Config.colorOn2[5] := 'off';
   instHMISettings.instAniPNTmr.stations.me[16].kp8Config.colorOn2[6] := 'off';
   instHMISettings.instAniPNTmr.stations.me[16].kp8Config.colorOff[0] := 'off';
   instHMISettings.instAniPNTmr.stations.me[16].kp8Config.colorOff[1] := 'off';
   instHMISettings.instAniPNTmr.stations.me[16].kp8Config.colorOff[2] := 'off';
   instHMISettings.instAniPNTmr.stations.me[16].kp8Config.colorOff[3] := 'green';
   instHMISettings.instAniPNTmr.stations.me[16].kp8Config.colorOff[4] := 'off';
   instHMISettings.instAniPNTmr.stations.me[16].kp8Config.colorOff[5] := 'off';
   instHMISettings.instAniPNTmr.stations.me[16].kp8Config.colorOff[6] := 'off';
   instHMISettings.instAniPNTmr.stations.me[16].kp8Config.colorOff[7] := 'green';
   instHMISettings.instAniPNTmr.stations.me[16].kp8Config.mode[3] := TRUE;
   instHMISettings.instAniPNTmr.stations.me[16].kp8Config.mode[7] := TRUE;
   instHMISettings.instAniPNTmr.stations.me[16].kp8Out := 16#0088_0000;
   instHMISettings.instAniPNTmr.stations.me[16].line := WSTRING#'CDO';
   instHMISettings.instAniPNTmr.stations.me[16].partNumbers[0] := WSTRING#'';
   instHMISettings.instAniPNTmr.stations.me[16].partNumbers[1] := WSTRING#'';
   instHMISettings.instAniPNTmr.stations.me[16].partNumbers[2] := WSTRING#'';
   instHMISettings.instAniPNTmr.stations.me[16].partNumbers[3] := WSTRING#'16.08.216.911.030B';
   instHMISettings.instAniPNTmr.stations.me[16].partNumbers[4] := WSTRING#'';
   instHMISettings.instAniPNTmr.stations.me[16].partNumbers[5] := WSTRING#'';
   instHMISettings.instAniPNTmr.stations.me[16].partNumbers[6] := WSTRING#'';
   instHMISettings.instAniPNTmr.stations.me[16].partNumbers[7] := WSTRING#'16.08.216.912.050A';
   instHMISettings.instAniPNTmr.stations.me[16].presetTime.allotted[3] := 1800.0;
   instHMISettings.instAniPNTmr.stations.me[16].presetTime.allotted[6] := 1800.0;
   instHMISettings.instAniPNTmr.stations.me[16].presetTime.allotted[7] := 1800.0;
   instHMISettings.instAniPNTmr.stations.me[16].presetTime.critical[3] := 300.0;
   instHMISettings.instAniPNTmr.stations.me[16].presetTime.critical[6] := 300.0;
   instHMISettings.instAniPNTmr.stations.me[16].presetTime.critical[7] := 300.0;
   instHMISettings.instAniPNTmr.stations.me[16].stackLightOut := 16#2400_0000;
   instHMISettings.instAniPNTmr.stations.me[17].dropZone := 2;
   instHMISettings.instAniPNTmr.stations.me[17].kp8Config.activate[2] := TRUE;
   instHMISettings.instAniPNTmr.stations.me[17].kp8Config.activate[3] := TRUE;
   instHMISettings.instAniPNTmr.stations.me[17].kp8Config.activate[6] := TRUE;
   instHMISettings.instAniPNTmr.stations.me[17].kp8Config.activate[7] := TRUE;
   instHMISettings.instAniPNTmr.stations.me[17].kp8Config.colorOn1[0] := 'off';
   instHMISettings.instAniPNTmr.stations.me[17].kp8Config.colorOn1[1] := 'off';
   instHMISettings.instAniPNTmr.stations.me[17].kp8Config.colorOn1[2] := 'yellow';
   instHMISettings.instAniPNTmr.stations.me[17].kp8Config.colorOn1[3] := 'yellow';
   instHMISettings.instAniPNTmr.stations.me[17].kp8Config.colorOn1[4] := 'off';
   instHMISettings.instAniPNTmr.stations.me[17].kp8Config.colorOn1[5] := 'off';
   instHMISettings.instAniPNTmr.stations.me[17].kp8Config.colorOn1[6] := 'yellow';
   instHMISettings.instAniPNTmr.stations.me[17].kp8Config.colorOn1[7] := 'yellow';
   instHMISettings.instAniPNTmr.stations.me[17].kp8Config.colorOn2[0] := 'off';
   instHMISettings.instAniPNTmr.stations.me[17].kp8Config.colorOn2[1] := 'off';
   instHMISettings.instAniPNTmr.stations.me[17].kp8Config.colorOn2[4] := 'off';
   instHMISettings.instAniPNTmr.stations.me[17].kp8Config.colorOn2[5] := 'off';
   instHMISettings.instAniPNTmr.stations.me[17].kp8Config.colorOff[0] := 'off';
   instHMISettings.instAniPNTmr.stations.me[17].kp8Config.colorOff[1] := 'off';
   instHMISettings.instAniPNTmr.stations.me[17].kp8Config.colorOff[2] := 'green';
   instHMISettings.instAniPNTmr.stations.me[17].kp8Config.colorOff[3] := 'green';
   instHMISettings.instAniPNTmr.stations.me[17].kp8Config.colorOff[4] := 'off';
   instHMISettings.instAniPNTmr.stations.me[17].kp8Config.colorOff[5] := 'off';
   instHMISettings.instAniPNTmr.stations.me[17].kp8Config.colorOff[6] := 'green';
   instHMISettings.instAniPNTmr.stations.me[17].kp8Config.colorOff[7] := 'green';
   instHMISettings.instAniPNTmr.stations.me[17].kp8Config.mode[2] := TRUE;
   instHMISettings.instAniPNTmr.stations.me[17].kp8Config.mode[3] := TRUE;
   instHMISettings.instAniPNTmr.stations.me[17].kp8Config.mode[6] := TRUE;
   instHMISettings.instAniPNTmr.stations.me[17].kp8Config.mode[7] := TRUE;
   instHMISettings.instAniPNTmr.stations.me[17].kp8Out := 16#00CC_0000;
   instHMISettings.instAniPNTmr.stations.me[17].line := WSTRING#'CDO';
   instHMISettings.instAniPNTmr.stations.me[17].partNumbers[0] := WSTRING#'';
   instHMISettings.instAniPNTmr.stations.me[17].partNumbers[1] := WSTRING#'';
   instHMISettings.instAniPNTmr.stations.me[17].partNumbers[2] := WSTRING#'16.08.216.790.001A';
   instHMISettings.instAniPNTmr.stations.me[17].partNumbers[3] := WSTRING#'16.08.208.691.010D';
   instHMISettings.instAniPNTmr.stations.me[17].partNumbers[4] := WSTRING#'';
   instHMISettings.instAniPNTmr.stations.me[17].partNumbers[5] := WSTRING#'';
   instHMISettings.instAniPNTmr.stations.me[17].partNumbers[6] := WSTRING#'16.08.216.501.010A';
   instHMISettings.instAniPNTmr.stations.me[17].partNumbers[7] := WSTRING#'16.08.208.531.020L';
   instHMISettings.instAniPNTmr.stations.me[17].presetTime.allotted[2] := 1800.0;
   instHMISettings.instAniPNTmr.stations.me[17].presetTime.allotted[3] := 1800.0;
   instHMISettings.instAniPNTmr.stations.me[17].presetTime.allotted[6] := 1800.0;
   instHMISettings.instAniPNTmr.stations.me[17].presetTime.allotted[7] := 1800.0;
   instHMISettings.instAniPNTmr.stations.me[17].presetTime.critical[2] := 300.0;
   instHMISettings.instAniPNTmr.stations.me[17].presetTime.critical[3] := 300.0;
   instHMISettings.instAniPNTmr.stations.me[17].presetTime.critical[6] := 300.0;
   instHMISettings.instAniPNTmr.stations.me[17].presetTime.critical[7] := 300.0;
   instHMISettings.instAniPNTmr.stations.me[17].stackLightOut := 16#2409_0000;
   instHMISettings.instAniPNTmr.stations.me[18].dropZone := 3;
   instHMISettings.instAniPNTmr.stations.me[18].kp8Config.activate[3] := TRUE;
   instHMISettings.instAniPNTmr.stations.me[18].kp8Config.activate[6] := TRUE;
   instHMISettings.instAniPNTmr.stations.me[18].kp8Config.activate[7] := TRUE;
   instHMISettings.instAniPNTmr.stations.me[18].kp8Config.colorOn1[0] := 'off';
   instHMISettings.instAniPNTmr.stations.me[18].kp8Config.colorOn1[1] := 'off';
   instHMISettings.instAniPNTmr.stations.me[18].kp8Config.colorOn1[2] := 'off';
   instHMISettings.instAniPNTmr.stations.me[18].kp8Config.colorOn1[3] := 'yellow';
   instHMISettings.instAniPNTmr.stations.me[18].kp8Config.colorOn1[4] := 'off';
   instHMISettings.instAniPNTmr.stations.me[18].kp8Config.colorOn1[5] := 'off';
   instHMISettings.instAniPNTmr.stations.me[18].kp8Config.colorOn1[6] := 'yellow';
   instHMISettings.instAniPNTmr.stations.me[18].kp8Config.colorOn1[7] := 'yellow';
   instHMISettings.instAniPNTmr.stations.me[18].kp8Config.colorOn2[0] := 'off';
   instHMISettings.instAniPNTmr.stations.me[18].kp8Config.colorOn2[1] := 'off';
   instHMISettings.instAniPNTmr.stations.me[18].kp8Config.colorOn2[2] := 'off';
   instHMISettings.instAniPNTmr.stations.me[18].kp8Config.colorOn2[4] := 'off';
   instHMISettings.instAniPNTmr.stations.me[18].kp8Config.colorOn2[5] := 'off';
   instHMISettings.instAniPNTmr.stations.me[18].kp8Config.colorOff[0] := 'off';
   instHMISettings.instAniPNTmr.stations.me[18].kp8Config.colorOff[1] := 'off';
   instHMISettings.instAniPNTmr.stations.me[18].kp8Config.colorOff[2] := 'off';
   instHMISettings.instAniPNTmr.stations.me[18].kp8Config.colorOff[3] := 'green';
   instHMISettings.instAniPNTmr.stations.me[18].kp8Config.colorOff[4] := 'off';
   instHMISettings.instAniPNTmr.stations.me[18].kp8Config.colorOff[5] := 'off';
   instHMISettings.instAniPNTmr.stations.me[18].kp8Config.colorOff[6] := 'green';
   instHMISettings.instAniPNTmr.stations.me[18].kp8Config.colorOff[7] := 'green';
   instHMISettings.instAniPNTmr.stations.me[18].kp8Config.mode[3] := TRUE;
   instHMISettings.instAniPNTmr.stations.me[18].kp8Config.mode[6] := TRUE;
   instHMISettings.instAniPNTmr.stations.me[18].kp8Config.mode[7] := TRUE;
   instHMISettings.instAniPNTmr.stations.me[18].kp8Out := 16#00C8_0000;
   instHMISettings.instAniPNTmr.stations.me[18].line := WSTRING#'CDO';
   instHMISettings.instAniPNTmr.stations.me[18].partNumbers[0] := WSTRING#'';
   instHMISettings.instAniPNTmr.stations.me[18].partNumbers[1] := WSTRING#'';
   instHMISettings.instAniPNTmr.stations.me[18].partNumbers[2] := WSTRING#'';
   instHMISettings.instAniPNTmr.stations.me[18].partNumbers[3] := WSTRING#'16.08.208.331.000F';
   instHMISettings.instAniPNTmr.stations.me[18].partNumbers[4] := WSTRING#'';
   instHMISettings.instAniPNTmr.stations.me[18].partNumbers[5] := WSTRING#'';
   instHMISettings.instAniPNTmr.stations.me[18].partNumbers[6] := WSTRING#'16.08.216.181.020A';
   instHMISettings.instAniPNTmr.stations.me[18].partNumbers[7] := WSTRING#'16.08.216.951.010A';
   instHMISettings.instAniPNTmr.stations.me[18].presetTime.allotted[3] := 1800.0;
   instHMISettings.instAniPNTmr.stations.me[18].presetTime.allotted[6] := 1800.0;
   instHMISettings.instAniPNTmr.stations.me[18].presetTime.allotted[7] := 1800.0;
   instHMISettings.instAniPNTmr.stations.me[18].presetTime.critical[3] := 300.0;
   instHMISettings.instAniPNTmr.stations.me[18].presetTime.critical[6] := 300.0;
   instHMISettings.instAniPNTmr.stations.me[18].presetTime.critical[7] := 300.0;
   instHMISettings.instAniPNTmr.stations.me[18].stackLightOut := 16#2401_0000;
   instHMISettings.instAniPNTmr.stations.me[19].dropZone := 1;
   instHMISettings.instAniPNTmr.stations.me[19].kp8Config.activate[1] := TRUE;
   instHMISettings.instAniPNTmr.stations.me[19].kp8Config.activate[2] := TRUE;
   instHMISettings.instAniPNTmr.stations.me[19].kp8Config.activate[3] := TRUE;
   instHMISettings.instAniPNTmr.stations.me[19].kp8Config.activate[5] := TRUE;
   instHMISettings.instAniPNTmr.stations.me[19].kp8Config.activate[6] := TRUE;
   instHMISettings.instAniPNTmr.stations.me[19].kp8Config.activate[7] := TRUE;
   instHMISettings.instAniPNTmr.stations.me[19].kp8Config.colorOn1[0] := 'off';
   instHMISettings.instAniPNTmr.stations.me[19].kp8Config.colorOn1[1] := 'yellow';
   instHMISettings.instAniPNTmr.stations.me[19].kp8Config.colorOn1[2] := 'yellow';
   instHMISettings.instAniPNTmr.stations.me[19].kp8Config.colorOn1[3] := 'yellow';
   instHMISettings.instAniPNTmr.stations.me[19].kp8Config.colorOn1[4] := 'off';
   instHMISettings.instAniPNTmr.stations.me[19].kp8Config.colorOn1[5] := 'yellow';
   instHMISettings.instAniPNTmr.stations.me[19].kp8Config.colorOn1[6] := 'yellow';
   instHMISettings.instAniPNTmr.stations.me[19].kp8Config.colorOn1[7] := 'yellow';
   instHMISettings.instAniPNTmr.stations.me[19].kp8Config.colorOn2[0] := 'off';
   instHMISettings.instAniPNTmr.stations.me[19].kp8Config.colorOn2[4] := 'off';
   instHMISettings.instAniPNTmr.stations.me[19].kp8Config.colorOff[0] := 'off';
   instHMISettings.instAniPNTmr.stations.me[19].kp8Config.colorOff[1] := 'green';
   instHMISettings.instAniPNTmr.stations.me[19].kp8Config.colorOff[2] := 'green';
   instHMISettings.instAniPNTmr.stations.me[19].kp8Config.colorOff[3] := 'green';
   instHMISettings.instAniPNTmr.stations.me[19].kp8Config.colorOff[4] := 'off';
   instHMISettings.instAniPNTmr.stations.me[19].kp8Config.colorOff[5] := 'green';
   instHMISettings.instAniPNTmr.stations.me[19].kp8Config.colorOff[6] := 'green';
   instHMISettings.instAniPNTmr.stations.me[19].kp8Config.colorOff[7] := 'green';
   instHMISettings.instAniPNTmr.stations.me[19].kp8Config.mode[1] := TRUE;
   instHMISettings.instAniPNTmr.stations.me[19].kp8Config.mode[2] := TRUE;
   instHMISettings.instAniPNTmr.stations.me[19].kp8Config.mode[3] := TRUE;
   instHMISettings.instAniPNTmr.stations.me[19].kp8Config.mode[5] := TRUE;
   instHMISettings.instAniPNTmr.stations.me[19].kp8Config.mode[6] := TRUE;
   instHMISettings.instAniPNTmr.stations.me[19].kp8Config.mode[7] := TRUE;
   instHMISettings.instAniPNTmr.stations.me[19].kp8Out := 16#00EE_0000;
   instHMISettings.instAniPNTmr.stations.me[19].line := WSTRING#'BFL';
   instHMISettings.instAniPNTmr.stations.me[19].partNumbers[0] := WSTRING#'';
   instHMISettings.instAniPNTmr.stations.me[19].partNumbers[1] := WSTRING#'16.08.216.521.000F';
   instHMISettings.instAniPNTmr.stations.me[19].partNumbers[2] := WSTRING#'16.08.216.831.020A';
   instHMISettings.instAniPNTmr.stations.me[19].partNumbers[3] := WSTRING#'16.08.208.151.010F';
   instHMISettings.instAniPNTmr.stations.me[19].partNumbers[4] := WSTRING#'';
   instHMISettings.instAniPNTmr.stations.me[19].partNumbers[5] := WSTRING#'16.08.217.411.080A';
   instHMISettings.instAniPNTmr.stations.me[19].partNumbers[6] := WSTRING#'16.08.216.151.010B';
   instHMISettings.instAniPNTmr.stations.me[19].partNumbers[7] := WSTRING#'16.08.211.511.020F';
   instHMISettings.instAniPNTmr.stations.me[19].presetTime.allotted[1] := 1800.0;
   instHMISettings.instAniPNTmr.stations.me[19].presetTime.allotted[2] := 1800.0;
   instHMISettings.instAniPNTmr.stations.me[19].presetTime.allotted[3] := 1800.0;
   instHMISettings.instAniPNTmr.stations.me[19].presetTime.allotted[5] := 120.0;
   instHMISettings.instAniPNTmr.stations.me[19].presetTime.allotted[6] := 1800.0;
   instHMISettings.instAniPNTmr.stations.me[19].presetTime.allotted[7] := 1800.0;
   instHMISettings.instAniPNTmr.stations.me[19].presetTime.critical[1] := 300.0;
   instHMISettings.instAniPNTmr.stations.me[19].presetTime.critical[2] := 300.0;
   instHMISettings.instAniPNTmr.stations.me[19].presetTime.critical[3] := 300.0;
   instHMISettings.instAniPNTmr.stations.me[19].presetTime.critical[5] := 70.0;
   instHMISettings.instAniPNTmr.stations.me[19].presetTime.critical[6] := 300.0;
   instHMISettings.instAniPNTmr.stations.me[19].presetTime.critical[7] := 300.0;
   instHMISettings.instAniPNTmr.stations.me[19].settings.selected := TRUE;
   instHMISettings.instAniPNTmr.stations.me[19].stackLightOut := 16#2449_0200;
   instHMISettings.instAniPNTmr.stations.me[20].dropZone := 2;
   instHMISettings.instAniPNTmr.stations.me[20].kp8Config.colorOn1[0] := 'off';
   instHMISettings.instAniPNTmr.stations.me[20].kp8Config.colorOn1[1] := 'off';
   instHMISettings.instAniPNTmr.stations.me[20].kp8Config.colorOn1[2] := 'off';
   instHMISettings.instAniPNTmr.stations.me[20].kp8Config.colorOn1[3] := 'off';
   instHMISettings.instAniPNTmr.stations.me[20].kp8Config.colorOn1[4] := 'off';
   instHMISettings.instAniPNTmr.stations.me[20].kp8Config.colorOn1[5] := 'off';
   instHMISettings.instAniPNTmr.stations.me[20].kp8Config.colorOn1[6] := 'off';
   instHMISettings.instAniPNTmr.stations.me[20].kp8Config.colorOn1[7] := 'off';
   instHMISettings.instAniPNTmr.stations.me[20].kp8Config.colorOn2[0] := 'off';
   instHMISettings.instAniPNTmr.stations.me[20].kp8Config.colorOn2[1] := 'off';
   instHMISettings.instAniPNTmr.stations.me[20].kp8Config.colorOn2[2] := 'off';
   instHMISettings.instAniPNTmr.stations.me[20].kp8Config.colorOn2[3] := 'off';
   instHMISettings.instAniPNTmr.stations.me[20].kp8Config.colorOn2[4] := 'off';
   instHMISettings.instAniPNTmr.stations.me[20].kp8Config.colorOn2[5] := 'off';
   instHMISettings.instAniPNTmr.stations.me[20].kp8Config.colorOn2[6] := 'off';
   instHMISettings.instAniPNTmr.stations.me[20].kp8Config.colorOn2[7] := 'off';
   instHMISettings.instAniPNTmr.stations.me[20].kp8Config.colorOff[0] := 'off';
   instHMISettings.instAniPNTmr.stations.me[20].kp8Config.colorOff[1] := 'off';
   instHMISettings.instAniPNTmr.stations.me[20].kp8Config.colorOff[2] := 'off';
   instHMISettings.instAniPNTmr.stations.me[20].kp8Config.colorOff[3] := 'off';
   instHMISettings.instAniPNTmr.stations.me[20].kp8Config.colorOff[4] := 'off';
   instHMISettings.instAniPNTmr.stations.me[20].kp8Config.colorOff[5] := 'off';
   instHMISettings.instAniPNTmr.stations.me[20].kp8Config.colorOff[6] := 'off';
   instHMISettings.instAniPNTmr.stations.me[20].kp8Config.colorOff[7] := 'off';
   instHMISettings.instAniPNTmr.stations.me[20].kp8Out := 16#0000_0000;
   instHMISettings.instAniPNTmr.stations.me[20].line := WSTRING#'BFL';
   instHMISettings.instAniPNTmr.stations.me[20].partNumbers[0] := WSTRING#'';
   instHMISettings.instAniPNTmr.stations.me[20].partNumbers[1] := WSTRING#'';
   instHMISettings.instAniPNTmr.stations.me[20].partNumbers[2] := WSTRING#'';
   instHMISettings.instAniPNTmr.stations.me[20].partNumbers[3] := WSTRING#'';
   instHMISettings.instAniPNTmr.stations.me[20].partNumbers[4] := WSTRING#'';
   instHMISettings.instAniPNTmr.stations.me[20].partNumbers[5] := WSTRING#'';
   instHMISettings.instAniPNTmr.stations.me[20].partNumbers[6] := WSTRING#'';
   instHMISettings.instAniPNTmr.stations.me[20].partNumbers[7] := WSTRING#'';
   instHMISettings.instAniPNTmr.stations.me[20].stackLightOut := 16#0000_0000;
   instHMISettings.instAniPNTmr.stations.me[21].dropZone := 3;
   instHMISettings.instAniPNTmr.stations.me[21].kp8Config.activate[7] := TRUE;
   instHMISettings.instAniPNTmr.stations.me[21].kp8Config.colorOn1[0] := 'off';
   instHMISettings.instAniPNTmr.stations.me[21].kp8Config.colorOn1[1] := 'off';
   instHMISettings.instAniPNTmr.stations.me[21].kp8Config.colorOn1[2] := 'off';
   instHMISettings.instAniPNTmr.stations.me[21].kp8Config.colorOn1[3] := 'off';
   instHMISettings.instAniPNTmr.stations.me[21].kp8Config.colorOn1[4] := 'off';
   instHMISettings.instAniPNTmr.stations.me[21].kp8Config.colorOn1[5] := 'off';
   instHMISettings.instAniPNTmr.stations.me[21].kp8Config.colorOn1[6] := 'off';
   instHMISettings.instAniPNTmr.stations.me[21].kp8Config.colorOn1[7] := 'yellow';
   instHMISettings.instAniPNTmr.stations.me[21].kp8Config.colorOn2[0] := 'off';
   instHMISettings.instAniPNTmr.stations.me[21].kp8Config.colorOn2[1] := 'off';
   instHMISettings.instAniPNTmr.stations.me[21].kp8Config.colorOn2[2] := 'off';
   instHMISettings.instAniPNTmr.stations.me[21].kp8Config.colorOn2[3] := 'off';
   instHMISettings.instAniPNTmr.stations.me[21].kp8Config.colorOn2[4] := 'off';
   instHMISettings.instAniPNTmr.stations.me[21].kp8Config.colorOn2[5] := 'off';
   instHMISettings.instAniPNTmr.stations.me[21].kp8Config.colorOn2[6] := 'off';
   instHMISettings.instAniPNTmr.stations.me[21].kp8Config.colorOff[0] := 'off';
   instHMISettings.instAniPNTmr.stations.me[21].kp8Config.colorOff[1] := 'off';
   instHMISettings.instAniPNTmr.stations.me[21].kp8Config.colorOff[2] := 'off';
   instHMISettings.instAniPNTmr.stations.me[21].kp8Config.colorOff[3] := 'off';
   instHMISettings.instAniPNTmr.stations.me[21].kp8Config.colorOff[4] := 'off';
   instHMISettings.instAniPNTmr.stations.me[21].kp8Config.colorOff[5] := 'off';
   instHMISettings.instAniPNTmr.stations.me[21].kp8Config.colorOff[6] := 'off';
   instHMISettings.instAniPNTmr.stations.me[21].kp8Config.colorOff[7] := 'green';
   instHMISettings.instAniPNTmr.stations.me[21].kp8Config.mode[7] := TRUE;
   instHMISettings.instAniPNTmr.stations.me[21].kp8Out := 16#0080_0000;
   instHMISettings.instAniPNTmr.stations.me[21].line := WSTRING#'BFL';
   instHMISettings.instAniPNTmr.stations.me[21].partNumbers[0] := WSTRING#'';
   instHMISettings.instAniPNTmr.stations.me[21].partNumbers[1] := WSTRING#'';
   instHMISettings.instAniPNTmr.stations.me[21].partNumbers[2] := WSTRING#'';
   instHMISettings.instAniPNTmr.stations.me[21].partNumbers[3] := WSTRING#'';
   instHMISettings.instAniPNTmr.stations.me[21].partNumbers[4] := WSTRING#'';
   instHMISettings.instAniPNTmr.stations.me[21].partNumbers[5] := WSTRING#'';
   instHMISettings.instAniPNTmr.stations.me[21].partNumbers[6] := WSTRING#'';
   instHMISettings.instAniPNTmr.stations.me[21].partNumbers[7] := WSTRING#'16.08.208.011.010G';
   instHMISettings.instAniPNTmr.stations.me[21].presetTime.allotted[7] := 1800.0;
   instHMISettings.instAniPNTmr.stations.me[21].presetTime.critical[7] := 300.0;
   instHMISettings.instAniPNTmr.stations.me[21].stackLightOut := 16#0400_0000;
   instHMISettings.instAniPNTmr.stations.me[22].dropZone := 1;
   instHMISettings.instAniPNTmr.stations.me[22].kp8Config.activate[3] := TRUE;
   instHMISettings.instAniPNTmr.stations.me[22].kp8Config.activate[6] := TRUE;
   instHMISettings.instAniPNTmr.stations.me[22].kp8Config.activate[7] := TRUE;
   instHMISettings.instAniPNTmr.stations.me[22].kp8Config.colorOn1[0] := 'off';
   instHMISettings.instAniPNTmr.stations.me[22].kp8Config.colorOn1[1] := 'off';
   instHMISettings.instAniPNTmr.stations.me[22].kp8Config.colorOn1[2] := 'off';
   instHMISettings.instAniPNTmr.stations.me[22].kp8Config.colorOn1[3] := 'yellow';
   instHMISettings.instAniPNTmr.stations.me[22].kp8Config.colorOn1[4] := 'off';
   instHMISettings.instAniPNTmr.stations.me[22].kp8Config.colorOn1[5] := 'off';
   instHMISettings.instAniPNTmr.stations.me[22].kp8Config.colorOn1[6] := 'yellow';
   instHMISettings.instAniPNTmr.stations.me[22].kp8Config.colorOn1[7] := 'yellow';
   instHMISettings.instAniPNTmr.stations.me[22].kp8Config.colorOn2[0] := 'off';
   instHMISettings.instAniPNTmr.stations.me[22].kp8Config.colorOn2[1] := 'off';
   instHMISettings.instAniPNTmr.stations.me[22].kp8Config.colorOn2[2] := 'off';
   instHMISettings.instAniPNTmr.stations.me[22].kp8Config.colorOn2[4] := 'off';
   instHMISettings.instAniPNTmr.stations.me[22].kp8Config.colorOn2[5] := 'off';
   instHMISettings.instAniPNTmr.stations.me[22].kp8Config.colorOff[0] := 'off';
   instHMISettings.instAniPNTmr.stations.me[22].kp8Config.colorOff[1] := 'off';
   instHMISettings.instAniPNTmr.stations.me[22].kp8Config.colorOff[2] := 'off';
   instHMISettings.instAniPNTmr.stations.me[22].kp8Config.colorOff[3] := 'green';
   instHMISettings.instAniPNTmr.stations.me[22].kp8Config.colorOff[4] := 'off';
   instHMISettings.instAniPNTmr.stations.me[22].kp8Config.colorOff[5] := 'off';
   instHMISettings.instAniPNTmr.stations.me[22].kp8Config.colorOff[6] := 'green';
   instHMISettings.instAniPNTmr.stations.me[22].kp8Config.colorOff[7] := 'green';
   instHMISettings.instAniPNTmr.stations.me[22].kp8Config.mode[3] := TRUE;
   instHMISettings.instAniPNTmr.stations.me[22].kp8Config.mode[6] := TRUE;
   instHMISettings.instAniPNTmr.stations.me[22].kp8Config.mode[7] := TRUE;
   instHMISettings.instAniPNTmr.stations.me[22].kp8Out := 16#00C8_0000;
   instHMISettings.instAniPNTmr.stations.me[22].line := WSTRING#'LGS';
   instHMISettings.instAniPNTmr.stations.me[22].partNumbers[0] := WSTRING#'';
   instHMISettings.instAniPNTmr.stations.me[22].partNumbers[1] := WSTRING#'';
   instHMISettings.instAniPNTmr.stations.me[22].partNumbers[2] := WSTRING#'';
   instHMISettings.instAniPNTmr.stations.me[22].partNumbers[3] := WSTRING#'16.08.208.161.020F';
   instHMISettings.instAniPNTmr.stations.me[22].partNumbers[4] := WSTRING#'';
   instHMISettings.instAniPNTmr.stations.me[22].partNumbers[5] := WSTRING#'';
   instHMISettings.instAniPNTmr.stations.me[22].partNumbers[6] := WSTRING#'16.08.211.121.000G';
   instHMISettings.instAniPNTmr.stations.me[22].partNumbers[7] := WSTRING#'16.08.216.161.020A';
   instHMISettings.instAniPNTmr.stations.me[22].presetTime.allotted[3] := 1800.0;
   instHMISettings.instAniPNTmr.stations.me[22].presetTime.allotted[6] := 1800.0;
   instHMISettings.instAniPNTmr.stations.me[22].presetTime.allotted[7] := 1800.0;
   instHMISettings.instAniPNTmr.stations.me[22].presetTime.critical[3] := 300.0;
   instHMISettings.instAniPNTmr.stations.me[22].presetTime.critical[6] := 300.0;
   instHMISettings.instAniPNTmr.stations.me[22].presetTime.critical[7] := 300.0;
   instHMISettings.instAniPNTmr.stations.me[22].stackLightOut := 16#2401_0000;
   instHMISettings.instAniPNTmr.stations.me[23].dropZone := 2;
   instHMISettings.instAniPNTmr.stations.me[23].kp8Config.activate[7] := TRUE;
   instHMISettings.instAniPNTmr.stations.me[23].kp8Config.colorOn1[0] := 'off';
   instHMISettings.instAniPNTmr.stations.me[23].kp8Config.colorOn1[1] := 'off';
   instHMISettings.instAniPNTmr.stations.me[23].kp8Config.colorOn1[2] := 'off';
   instHMISettings.instAniPNTmr.stations.me[23].kp8Config.colorOn1[3] := 'off';
   instHMISettings.instAniPNTmr.stations.me[23].kp8Config.colorOn1[4] := 'off';
   instHMISettings.instAniPNTmr.stations.me[23].kp8Config.colorOn1[5] := 'off';
   instHMISettings.instAniPNTmr.stations.me[23].kp8Config.colorOn1[6] := 'off';
   instHMISettings.instAniPNTmr.stations.me[23].kp8Config.colorOn1[7] := 'yellow';
   instHMISettings.instAniPNTmr.stations.me[23].kp8Config.colorOn2[0] := 'off';
   instHMISettings.instAniPNTmr.stations.me[23].kp8Config.colorOn2[1] := 'off';
   instHMISettings.instAniPNTmr.stations.me[23].kp8Config.colorOn2[2] := 'off';
   instHMISettings.instAniPNTmr.stations.me[23].kp8Config.colorOn2[3] := 'off';
   instHMISettings.instAniPNTmr.stations.me[23].kp8Config.colorOn2[4] := 'off';
   instHMISettings.instAniPNTmr.stations.me[23].kp8Config.colorOn2[5] := 'off';
   instHMISettings.instAniPNTmr.stations.me[23].kp8Config.colorOn2[6] := 'off';
   instHMISettings.instAniPNTmr.stations.me[23].kp8Config.colorOff[0] := 'off';
   instHMISettings.instAniPNTmr.stations.me[23].kp8Config.colorOff[1] := 'off';
   instHMISettings.instAniPNTmr.stations.me[23].kp8Config.colorOff[2] := 'off';
   instHMISettings.instAniPNTmr.stations.me[23].kp8Config.colorOff[3] := 'off';
   instHMISettings.instAniPNTmr.stations.me[23].kp8Config.colorOff[4] := 'off';
   instHMISettings.instAniPNTmr.stations.me[23].kp8Config.colorOff[5] := 'off';
   instHMISettings.instAniPNTmr.stations.me[23].kp8Config.colorOff[6] := 'off';
   instHMISettings.instAniPNTmr.stations.me[23].kp8Config.colorOff[7] := 'green';
   instHMISettings.instAniPNTmr.stations.me[23].kp8Config.mode[7] := TRUE;
   instHMISettings.instAniPNTmr.stations.me[23].kp8Out := 16#0080_0000;
   instHMISettings.instAniPNTmr.stations.me[23].line := WSTRING#'LGS';
   instHMISettings.instAniPNTmr.stations.me[23].partNumbers[0] := WSTRING#'';
   instHMISettings.instAniPNTmr.stations.me[23].partNumbers[1] := WSTRING#'';
   instHMISettings.instAniPNTmr.stations.me[23].partNumbers[2] := WSTRING#'';
   instHMISettings.instAniPNTmr.stations.me[23].partNumbers[3] := WSTRING#'';
   instHMISettings.instAniPNTmr.stations.me[23].partNumbers[4] := WSTRING#'';
   instHMISettings.instAniPNTmr.stations.me[23].partNumbers[5] := WSTRING#'';
   instHMISettings.instAniPNTmr.stations.me[23].partNumbers[6] := WSTRING#'';
   instHMISettings.instAniPNTmr.stations.me[23].partNumbers[7] := WSTRING#'16.08.208.021.020C';
   instHMISettings.instAniPNTmr.stations.me[23].presetTime.allotted[7] := 1800.0;
   instHMISettings.instAniPNTmr.stations.me[23].presetTime.critical[7] := 300.0;
   instHMISettings.instAniPNTmr.stations.me[23].stackLightOut := 16#0400_0000;
   instHMISettings.instAniPNTmr.stations.me[24].dropZone := 3;
   instHMISettings.instAniPNTmr.stations.me[24].kp8Config.activate[7] := TRUE;
